LIN {X 0,Y 310.174,Z 752.952,A -85,B 0,C 180,E1 -16266.197,E2 -16266.197} C_VEL
LIN {X 0,Y 308.581,Z 766.008,A -85,B 0,C 180,E1 -16267.045,E2 -16267.045} C_VEL
LIN {X 0,Y 306.78,Z 778.403,A -85,B 0,C 180,E1 -16268.145,E2 -16268.145} C_VEL
LIN {X 0,Y 304.905,Z 789.628,A -85,B 0,C 180,E1 -16269.421,E2 -16269.421} C_VEL
LIN {X 0,Y 302.875,Z 800.82,A -85,B 0,C 180,E1 -16271.043,E2 -16271.043} C_VEL
LIN {X 0,Y 301.234,Z 810.089,A -85,B 0,C 180,E1 -16272.722,E2 -16272.722} C_VEL
LIN {X 0,Y 299.736,Z 818.952,A -85,B 0,C 180,E1 -16274.706,E2 -16274.706} C_VEL
LIN {X 0,Y 298.426,Z 826.179,A -85,B 0,C 180,E1 -16276.726,E2 -16276.726} C_VEL
LIN {X 0,Y 297.408,Z 832.88,A -85,B 0,C 180,E1 -16279.103,E2 -16279.103} C_VEL
LIN {X 0,Y 297.02,Z 837.35,A -85,B 0,C 180,E1 -16281.153,E2 -16281.153} C_VEL
LIN {X 0,Y 296.852,Z 840.748,A -85,B 0,C 180,E1 -16283.202,E2 -16283.202} C_VEL
LIN {X 0,Y 296.856,Z 842.474,A -85,B 0,C 180,E1 -16284.566,E2 -16284.566} C_VEL
LIN {X 0,Y 296.874,Z 843.732,A -85,B 0,C 180,E1 -16285.928,E2 -16285.928} C_VEL
LIN {X 0,Y 297.025,Z 844.574,A -85,B 0,C 180,E1 -16287.288,E2 -16287.288} C_VEL
LIN {X 0,Y 297.158,Z 845.011,A -85,B 0,C 180,E1 -16288.645,E2 -16288.645} C_VEL
LIN {X 0,Y 297.234,Z 845.034,A -85,B 0,C 180,E1 -16290,E2 -16290} C_VEL
LIN {X 0,Y 297.191,Z 844.583,A -85,B 0,C 180,E1 -16291.355,E2 -16291.355} C_VEL
LIN {X 0,Y 296.924,Z 842.624,A -85,B 0,C 180,E1 -16294.072,E2 -16294.072} C_VEL
LIN {X 0,Y 296.873,Z 840.823,A -85,B 0,C 180,E1 -16296.128,E2 -16296.128} C_VEL
LIN {X 0,Y 296.997,Z 836.98,A -85,B 0,C 180,E1 -16298.848,E2 -16298.848} C_VEL
LIN {X 0,Y 297.414,Z 832.866,A -85,B 0,C 180,E1 -16300.897,E2 -16300.897} C_VEL
LIN {X 0,Y 298.462,Z 826.576,A -85,B 0,C 180,E1 -16303.272,E2 -16303.272} C_VEL
LIN {X 0,Y 299.734,Z 819.761,A -85,B 0,C 180,E1 -16305.294,E2 -16305.294} C_VEL
LIN {X 0,Y 301.187,Z 811.484,A -85,B 0,C 180,E1 -16307.273,E2 -16307.273} C_VEL
LIN {X 0,Y 302.982,Z 802.663,A -85,B 0,C 180,E1 -16308.95,E2 -16308.95} C_VEL
LIN {X 0,Y 305.047,Z 792.026,A -85,B 0,C 180,E1 -16310.569,E2 -16310.569} C_VEL
LIN {X 0,Y 306.884,Z 781.465,A -85,B 0,C 180,E1 -16311.847,E2 -16311.847} C_VEL
LIN {X 0,Y 308.764,Z 769.655,A -85,B 0,C 180,E1 -16312.941,E2 -16312.941} C_VEL
LIN {X 0,Y 310.313,Z 757.416,A -85,B 0,C 180,E1 -16313.791,E2 -16313.791} C_VEL
LIN {X 0,Y 311.486,Z 744.997,A -85,B 0,C 180,E1 -16314.397,E2 -16314.397} C_VEL
LIN {X 0,Y 312.109,Z 730.684,A -85,B 0,C 180,E1 -16314.824,E2 -16314.824} C_VEL
LIN {X 0,Y 313.469,Z 680.173,A -85,B 0,C 180,E1 -16316,E2 -16316} C_VEL
LIN {X 0,Y 310.399,Z 651.031,A -85,B 0,C 180,E1 -16317.095,E2 -16317.095} C_VEL
LIN {X 0,Y 306.302,Z 623.478,A -85,B 0,C 180,E1 -16318.301,E2 -16318.301} C_VEL
LIN {X 0,Y 305.071,Z 620.075,A -85,B 0,C 180,E1 -16318.539,E2 -16318.539} C_VEL
LIN {X 0,Y 303.666,Z 615.782,A -85,B 0,C 180,E1 -16318.956,E2 -16318.956} C_VEL
LIN {X 0,Y 300.127,Z 600.639,A -85,B 0,C 180,E1 -16322.586,E2 -16322.586} C_VEL
LIN {X 0,Y 298.408,Z 593.316,A -85,B 0,C 180,E1 -16324.418,E2 -16324.418} C_VEL
LIN {X 0,Y 298.438,Z 593.306,A -85,B 0,C 180,E1 -16327.753,E2 -16327.753} C_VEL
LIN {X 0,Y 298.418,Z 593.307,A -85,B 0,C 180,E1 -16331.255,E2 -16331.255} C_VEL
LIN {X 0,Y 298.414,Z 593.308,A -85,B 0,C 180,E1 -16334.952,E2 -16334.952} C_VEL
LIN {X 0,Y 298.448,Z 593.306,A -85,B 0,C 180,E1 -16338.749,E2 -16338.749} C_VEL
LIN {X 0,Y 298.466,Z 593.305,A -85,B 0,C 180,E1 -16343.185,E2 -16343.185} C_VEL
LIN {X 0,Y 298.393,Z 593.313,A -85,B 0,C 180,E1 -16347.199,E2 -16347.199} C_VEL
LIN {X 0,Y 298.427,Z 593.294,A -85,B 0,C 180,E1 -16350.614,E2 -16350.614} C_VEL
LIN {X 0,Y 298.479,Z 593.303,A -85,B 0,C 180,E1 -16353.474,E2 -16353.474} C_VEL
LIN {X 0,Y 298.428,Z 593.291,A -85,B 0,C 180,E1 -16356.697,E2 -16356.697} C_VEL
LIN {X 0,Y 298.533,Z 593.299,A -85,B 0,C 180,E1 -16360.756,E2 -16360.756} C_VEL
LIN {X 0,Y 298.586,Z 593.274,A -85,B 0,C 180,E1 -16364.994,E2 -16364.994} C_VEL
LIN {X 0,Y 298.584,Z 593.283,A -85,B 0,C 180,E1 -16369.146,E2 -16369.146} C_VEL
LIN {X 0,Y 298.734,Z 593.253,A -85,B 0,C 180,E1 -16371.885,E2 -16371.885} C_VEL
LIN {X 0,Y 298.654,Z 593.285,A -85,B 0,C 180,E1 -16374.599,E2 -16374.599} C_VEL
LIN {X 0,Y 298.918,Z 593.227,A -85,B 0,C 180,E1 -16378.653,E2 -16378.653} C_VEL
LIN {X 0,Y 298.92,Z 593.25,A -85,B 0,C 180,E1 -16381.347,E2 -16381.347} C_VEL
LIN {X 0,Y 298.652,Z 593.259,A -85,B 0,C 180,E1 -16385.401,E2 -16385.401} C_VEL
LIN {X 0,Y 298.748,Z 593.267,A -85,B 0,C 180,E1 -16388.114,E2 -16388.114} C_VEL
LIN {X 0,Y 298.545,Z 593.277,A -85,B 0,C 180,E1 -16392.232,E2 -16392.232} C_VEL
LIN {X 0,Y 298.6,Z 593.291,A -85,B 0,C 180,E1 -16395.209,E2 -16395.209} C_VEL
LIN {X 0,Y 298.533,Z 593.282,A -85,B 0,C 180,E1 -16399.244,E2 -16399.244} C_VEL
LIN {X 0,Y 298.451,Z 593.299,A -85,B 0,C 180,E1 -16403.598,E2 -16403.598} C_VEL
LIN {X 0,Y 298.484,Z 593.301,A -85,B 0,C 180,E1 -16406.575,E2 -16406.575} C_VEL
LIN {X 0,Y 298.417,Z 593.299,A -85,B 0,C 180,E1 -16409.642,E2 -16409.642} C_VEL
LIN {X 0,Y 298.393,Z 593.316,A -85,B 0,C 180,E1 -16412.801,E2 -16412.801} C_VEL
LIN {X 0,Y 298.461,Z 593.309,A -85,B 0,C 180,E1 -16416.813,E2 -16416.813} C_VEL
LIN {X 0,Y 298.414,Z 593.286,A -85,B 0,C 180,E1 -16421.095,E2 -16421.095} C_VEL
LIN {X 0,Y 298.385,Z 593.317,A -85,B 0,C 180,E1 -16424.959,E2 -16424.959} C_VEL
LIN {X 0,Y 298.384,Z 593.301,A -85,B 0,C 180,E1 -16428.826,E2 -16428.826} C_VEL
LIN {X 0,Y 299.45,Z 596.241,A -85,B 0,C 180,E1 -16429.063,E2 -16429.063} C_VEL
LIN {X 0,Y 300.765,Z 598.211,A -85,B 0,C 180,E1 -16429.286,E2 -16429.286} C_VEL
LIN {X 0,Y 309.42,Z 613.922,A -85,B 0,C 180,E1 -16430.763,E2 -16430.763} C_VEL
LIN {X 0,Y 315.519,Z 626.227,A -85,B 0,C 180,E1 -16431.769,E2 -16431.769} C_VEL
LIN {X 0,Y 313.772,Z 685.154,A -85,B 0,C 180,E1 -16433.117,E2 -16433.117} C_VEL
LIN {X 0,Y 313.31,Z 698.588,A -85,B 0,C 180,E1 -16433.58,E2 -16433.58} C_VEL
LIN {X 0,Y 312.556,Z 710.365,A -85,B 0,C 180,E1 -16434.225,E2 -16434.225} C_VEL
LIN {X 0,Y 311.19,Z 723.672,A -85,B 0,C 180,E1 -16435.233,E2 -16435.233} C_VEL
LIN {X 0,Y 309.686,Z 735.273,A -85,B 0,C 180,E1 -16436.417,E2 -16436.417} C_VEL
LIN {X 0,Y 307.85,Z 746.627,A -85,B 0,C 180,E1 -16437.903,E2 -16437.903} C_VEL
LIN {X 0,Y 306.244,Z 755.192,A -85,B 0,C 180,E1 -16439.296,E2 -16439.296} C_VEL
LIN {X 0,Y 304.567,Z 763.776,A -85,B 0,C 180,E1 -16441.016,E2 -16441.016} C_VEL
LIN {X 0,Y 302.719,Z 772.004,A -85,B 0,C 180,E1 -16443.083,E2 -16443.083} C_VEL
LIN {X 0,Y 301.166,Z 778.564,A -85,B 0,C 180,E1 -16445.163,E2 -16445.163} C_VEL
LIN {X 0,Y 299.918,Z 783.703,A -85,B 0,C 180,E1 -16447.255,E2 -16447.255} C_VEL
LIN {X 0,Y 298.942,Z 787.596,A -85,B 0,C 180,E1 -16449.351,E2 -16449.351} C_VEL
LIN {X 0,Y 298.401,Z 789.563,A -85,B 0,C 180,E1 -16450.748,E2 -16450.748} C_VEL
LIN {X 0,Y 297.93,Z 791.107,A -85,B 0,C 180,E1 -16452.142,E2 -16452.142} C_VEL
LIN {X 0,Y 297.608,Z 792.207,A -85,B 0,C 180,E1 -16453.538,E2 -16453.538} C_VEL
LIN {X 0,Y 297.279,Z 793.073,A -85,B 0,C 180,E1 -16455.763,E2 -16455.763} C_VEL
LIN {X 0,Y 297.101,Z 792.993,A -85,B 0,C 180,E1 -16457.708,E2 -16457.708} C_VEL
LIN {X 0,Y 297.138,Z 791.447,A -85,B 0,C 180,E1 -16460.47,E2 -16460.47} C_VEL
LIN {X 0,Y 297.472,Z 788.763,A -85,B 0,C 180,E1 -16462.878,E2 -16462.878} C_VEL
LIN {X 0,Y 297.889,Z 784.726,A -85,B 0,C 180,E1 -16465.264,E2 -16465.264} C_VEL
LIN {X 0,Y 298.386,Z 780.095,A -85,B 0,C 180,E1 -16467.3,E2 -16467.3} C_VEL
LIN {X 0,Y 299.358,Z 773.121,A -85,B 0,C 180,E1 -16469.664,E2 -16469.664} C_VEL
LIN {X 0,Y 300.322,Z 765.523,A -85,B 0,C 180,E1 -16471.676,E2 -16471.676} C_VEL
LIN {X 0,Y 301.652,Z 756.013,A -85,B 0,C 180,E1 -16473.673,E2 -16473.673} C_VEL
LIN {X 0,Y 302.841,Z 746.175,A -85,B 0,C 180,E1 -16475.326,E2 -16475.326} C_VEL
LIN {X 0,Y 304.074,Z 735.11,A -85,B 0,C 180,E1 -16476.803,E2 -16476.803} C_VEL
LIN {X 0,Y 305.201,Z 724.278,A -85,B 0,C 180,E1 -16477.941,E2 -16477.941} C_VEL
LIN {X 0,Y 306.119,Z 712.245,A -85,B 0,C 180,E1 -16478.915,E2 -16478.915} C_VEL
LIN {X 0,Y 306.772,Z 699.048,A -85,B 0,C 180,E1 -16479.685,E2 -16479.685} C_VEL
LIN {X 0,Y 307.167,Z 685.86,A -85,B 0,C 180,E1 -16480.172,E2 -16480.172} C_VEL
LIN {X 0,Y 308.638,Z 618.658,A -85,B 0,C 180,E1 -16481.718,E2 -16481.718} C_VEL
LIN {X 0,Y 300.49,Z 598.313,A -85,B 0,C 180,E1 -16482.804,E2 -16482.804} C_VEL
LIN {X 0,Y 298.671,Z 593.897,A -85,B 0,C 180,E1 -16483.051,E2 -16483.051} C_VEL
LIN {X 0,Y 298.573,Z 593.291,A -85,B 0,C 180,E1 -16483.105,E2 -16483.105} C_VEL
LIN {X 0,Y 298.55,Z 593.296,A -85,B 0,C 180,E1 -16486.408,E2 -16486.408} C_VEL
LIN {X 0,Y 298.489,Z 593.302,A -85,B 0,C 180,E1 -16490.42,E2 -16490.42} C_VEL
LIN {X 0,Y 300.198,Z 597.98,A -85,B 0,C 180,E1 -16490.715,E2 -16490.715} C_VEL
LIN {X 0,Y 309.443,Z 620.601,A -85,B 0,C 180,E1 -16492.025,E2 -16492.025} C_VEL
LIN {X 0,Y 307.444,Z 689.886,A -85,B 0,C 180,E1 -16493.812,E2 -16493.812} C_VEL
LIN {X 0,Y 306.954,Z 703.275,A -85,B 0,C 180,E1 -16494.428,E2 -16494.428} C_VEL
LIN {X 0,Y 306.073,Z 716.586,A -85,B 0,C 180,E1 -16495.319,E2 -16495.319} C_VEL
LIN {X 0,Y 304.967,Z 729.092,A -85,B 0,C 180,E1 -16496.464,E2 -16496.464} C_VEL
LIN {X 0,Y 303.873,Z 739.878,A -85,B 0,C 180,E1 -16497.727,E2 -16497.727} C_VEL
LIN {X 0,Y 302.694,Z 749.874,A -85,B 0,C 180,E1 -16499.181,E2 -16499.181} C_VEL
LIN {X 0,Y 301.405,Z 759.749,A -85,B 0,C 180,E1 -16500.97,E2 -16500.97} C_VEL
LIN {X 0,Y 300.209,Z 763.729,A -85,B 0,C 180,E1 -16501.773,E2 -16501.773} C_VEL
LIN {X 0,Y 296.521,Z 769.833,A -85,B 0,C 180,E1 -16503.098,E2 -16503.098} C_VEL
LIN {X 0,Y 292.936,Z 775.382,A -85,B 0,C 180,E1 -16504.541,E2 -16504.541} C_VEL
LIN {X 0,Y 291.921,Z 778.388,A -85,B 0,C 180,E1 -16505.513,E2 -16505.513} C_VEL
LIN {X 0,Y 291.307,Z 782.87,A -85,B 0,C 180,E1 -16507.236,E2 -16507.236} C_VEL
LIN {X 0,Y 290.716,Z 787.192,A -85,B 0,C 180,E1 -16509.322,E2 -16509.322} C_VEL
LIN {X 0,Y 290.298,Z 790.365,A -85,B 0,C 180,E1 -16511.366,E2 -16511.366} C_VEL
LIN {X 0,Y 290.027,Z 792.549,A -85,B 0,C 180,E1 -16513.367,E2 -16513.367} C_VEL
LIN {X 0,Y 289.944,Z 793.863,A -85,B 0,C 180,E1 -16515.337,E2 -16515.337} C_VEL
LIN {X 0,Y 290.001,Z 794.378,A -85,B 0,C 180,E1 -16517.268,E2 -16517.268} C_VEL
LIN {X 0,Y 290.247,Z 794.094,A -85,B 0,C 180,E1 -16519.173,E2 -16519.173} C_VEL
LIN {X 0,Y 290.641,Z 793.064,A -85,B 0,C 180,E1 -16521.045,E2 -16521.045} C_VEL
LIN {X 0,Y 291.526,Z 790.21,A -85,B 0,C 180,E1 -16523.798,E2 -16523.798} C_VEL
LIN {X 0,Y 292.255,Z 787.193,A -85,B 0,C 180,E1 -16525.704,E2 -16525.704} C_VEL
LIN {X 0,Y 293.568,Z 781.749,A -85,B 0,C 180,E1 -16528.219,E2 -16528.219} C_VEL
LIN {X 0,Y 295.07,Z 775.583,A -85,B 0,C 180,E1 -16530.376,E2 -16530.376} C_VEL
LIN {X 0,Y 296.803,Z 767.866,A -85,B 0,C 180,E1 -16532.5,E2 -16532.5} C_VEL
LIN {X 0,Y 298.563,Z 759.264,A -85,B 0,C 180,E1 -16534.371,E2 -16534.371} C_VEL
LIN {X 0,Y 300.443,Z 749.499,A -85,B 0,C 180,E1 -16536.072,E2 -16536.072} C_VEL
LIN {X 0,Y 302.011,Z 739.942,A -85,B 0,C 180,E1 -16537.421,E2 -16537.421} C_VEL
LIN {X 0,Y 303.469,Z 729.502,A -85,B 0,C 180,E1 -16538.608,E2 -16538.608} C_VEL
LIN {X 0,Y 304.841,Z 717.293,A -85,B 0,C 180,E1 -16539.68,E2 -16539.68} C_VEL
LIN {X 0,Y 305.897,Z 703.764,A -85,B 0,C 180,E1 -16540.56,E2 -16540.56} C_VEL
LIN {X 0,Y 306.53,Z 690.829,A -85,B 0,C 180,E1 -16541.111,E2 -16541.111} C_VEL
LIN {X 0,Y 309.007,Z 627.426,A -85,B 0,C 180,E1 -16542.841,E2 -16542.841} C_VEL
LIN {X 0,Y 302.168,Z 613.302,A -85,B 0,C 180,E1 -16544.183,E2 -16544.183} C_VEL
LIN {X 0,Y 295.467,Z 601.572,A -85,B 0,C 180,E1 -16545.544,E2 -16545.544} C_VEL
LIN {X 0,Y 293.449,Z 598.204,A -85,B 0,C 180,E1 -16545.968,E2 -16545.968} C_VEL
LIN {X 0,Y 291.914,Z 595.837,A -85,B 0,C 180,E1 -16546.291,E2 -16546.291} C_VEL
LIN {X 0,Y 291.511,Z 594.173,A -85,B 0,C 180,E1 -16546.449,E2 -16546.449} C_VEL
LIN {X 0,Y 291.699,Z 594.15,A -85,B 0,C 180,E1 -16551.041,E2 -16551.041} C_VEL
LIN {X 0,Y 291.741,Z 594.143,A -85,B 0,C 180,E1 -16553.082,E2 -16553.082} C_VEL
LIN {X 0,Y 291.884,Z 594.126,A -85,B 0,C 180,E1 -16558.62,E2 -16558.62} C_VEL
LIN {X 0,Y 291.884,Z 594.126,A -85,B 0,C 180,E1 -16561.38,E2 -16561.38} C_VEL
LIN {X 0,Y 291.737,Z 594.136,A -85,B 0,C 180,E1 -16566.918,E2 -16566.918} C_VEL
LIN {X 0,Y 291.623,Z 594.149,A -85,B 0,C 180,E1 -16569.712,E2 -16569.712} C_VEL
LIN {X 0,Y 291.516,Z 594.158,A -85,B 0,C 180,E1 -16573.951,E2 -16573.951} C_VEL
LIN {X 0,Y 291.48,Z 594.163,A -85,B 0,C 180,E1 -16576.818,E2 -16576.818} C_VEL
LIN {X 0,Y 291.445,Z 594.172,A -85,B 0,C 180,E1 -16579.875,E2 -16579.875} C_VEL
LIN {X 0,Y 291.394,Z 594.179,A -85,B 0,C 180,E1 -16584.206,E2 -16584.206} C_VEL
LIN {X 0,Y 291.417,Z 594.176,A -85,B 0,C 180,E1 -16587.272,E2 -16587.272} C_VEL
LIN {X 0,Y 291.333,Z 594.19,A -85,B 0,C 180,E1 -16590.437,E2 -16590.437} C_VEL
LIN {X 0,Y 291.34,Z 594.188,A -85,B 0,C 180,E1 -16593.699,E2 -16593.699} C_VEL
LIN {X 0,Y 291.401,Z 594.185,A -85,B 0,C 180,E1 -16597.262,E2 -16597.262} C_VEL
LIN {X 0,Y 291.397,Z 594.188,A -85,B 0,C 180,E1 -16600.632,E2 -16600.632} C_VEL
LIN {X 0,Y 291.35,Z 594.193,A -85,B 0,C 180,E1 -16604.391,E2 -16604.391} C_VEL
LIN {X 0,Y 291.355,Z 594.195,A -85,B 0,C 180,E1 -16608.398,E2 -16608.398} C_VEL
LIN {X 0,Y 291.421,Z 594.36,A -85,B 0,C 180,E1 -16609.452,E2 -16609.452} C_VEL
LIN {X 0,Y 294.286,Z 604.468,A -85,B 0,C 180,E1 -16613.343,E2 -16613.343} C_VEL
LIN {X 0,Y 296.493,Z 613.544,A -85,B 0,C 180,E1 -16616.466,E2 -16616.466} C_VEL
LIN {X 0,Y 298.475,Z 623.474,A -85,B 0,C 180,E1 -16619.587,E2 -16619.587} C_VEL
LIN {X 0,Y 298.861,Z 626.642,A -85,B 0,C 180,E1 -16620.5,E2 -16620.5} C_VEL
LIN {X 0,Y 302.721,Z 646.5,A -85,B 0,C 180,E1 -16621.678,E2 -16621.678} C_VEL
LIN {X 0,Y 305.472,Z 665.59,A -85,B 0,C 180,E1 -16622.639,E2 -16622.639} C_VEL
LIN {X 0,Y 307.206,Z 685.196,A -85,B 0,C 180,E1 -16623.471,E2 -16623.471} C_VEL
LIN {X 0,Y 305.129,Z 738.474,A -85,B 0,C 180,E1 -16624.925,E2 -16624.925} C_VEL
LIN {X 0,Y 303.993,Z 752.145,A -85,B 0,C 180,E1 -16625.546,E2 -16625.546} C_VEL
LIN {X 0,Y 302.391,Z 764.748,A -85,B 0,C 180,E1 -16626.365,E2 -16626.365} C_VEL
LIN {X 0,Y 300.505,Z 777.257,A -85,B 0,C 180,E1 -16627.483,E2 -16627.483} C_VEL
LIN {X 0,Y 298.517,Z 788.54,A -85,B 0,C 180,E1 -16628.779,E2 -16628.779} C_VEL
LIN {X 0,Y 296.585,Z 798.8,A -85,B 0,C 180,E1 -16630.265,E2 -16630.265} C_VEL
LIN {X 0,Y 294.742,Z 808.126,A -85,B 0,C 180,E1 -16631.942,E2 -16631.942} C_VEL
LIN {X 0,Y 293.161,Z 817.32,A -85,B 0,C 180,E1 -16633.997,E2 -16633.997} C_VEL
LIN {X 0,Y 291.686,Z 824.774,A -85,B 0,C 180,E1 -16636.058,E2 -16636.058} C_VEL
LIN {X 0,Y 290.629,Z 830.768,A -85,B 0,C 180,E1 -16638.139,E2 -16638.139} C_VEL
LIN {X 0,Y 290.064,Z 835.554,A -85,B 0,C 180,E1 -16640.235,E2 -16640.235} C_VEL
LIN {X 0,Y 289.808,Z 839.251,A -85,B 0,C 180,E1 -16642.335,E2 -16642.335} C_VEL
LIN {X 0,Y 289.768,Z 841.932,A -85,B 0,C 180,E1 -16644.433,E2 -16644.433} C_VEL
LIN {X 0,Y 289.801,Z 843.156,A -85,B 0,C 180,E1 -16645.828,E2 -16645.828} C_VEL
LIN {X 0,Y 289.931,Z 843.978,A -85,B 0,C 180,E1 -16647.221,E2 -16647.221} C_VEL
LIN {X 0,Y 290.095,Z 844.397,A -85,B 0,C 180,E1 -16648.612,E2 -16648.612} C_VEL
LIN {X 0,Y 290.169,Z 844.386,A -85,B 0,C 180,E1 -16650,E2 -16650} C_VEL
LIN {X 0,Y 290.13,Z 843.902,A -85,B 0,C 180,E1 -16651.388,E2 -16651.388} C_VEL
LIN {X 0,Y 289.847,Z 842.072,A -85,B 0,C 180,E1 -16654.171,E2 -16654.171} C_VEL
LIN {X 0,Y 289.782,Z 840.523,A -85,B 0,C 180,E1 -16656.085,E2 -16656.085} C_VEL
LIN {X 0,Y 289.846,Z 837.625,A -85,B 0,C 180,E1 -16658.365,E2 -16658.365} C_VEL
LIN {X 0,Y 290.201,Z 833.917,A -85,B 0,C 180,E1 -16660.465,E2 -16660.465} C_VEL
LIN {X 0,Y 290.962,Z 829.105,A -85,B 0,C 180,E1 -16662.555,E2 -16662.555} C_VEL
LIN {X 0,Y 292.076,Z 823.047,A -85,B 0,C 180,E1 -16664.634,E2 -16664.634} C_VEL
LIN {X 0,Y 293.602,Z 815.546,A -85,B 0,C 180,E1 -16666.693,E2 -16666.693} C_VEL
LIN {X 0,Y 295.098,Z 807.922,A -85,B 0,C 180,E1 -16668.394,E2 -16668.394} C_VEL
LIN {X 0,Y 297.092,Z 798.69,A -85,B 0,C 180,E1 -16670.06,E2 -16670.06} C_VEL
LIN {X 0,Y 299.166,Z 788.43,A -85,B 0,C 180,E1 -16671.534,E2 -16671.534} C_VEL
LIN {X 0,Y 301.092,Z 777.083,A -85,B 0,C 180,E1 -16672.833,E2 -16672.833} C_VEL
LIN {X 0,Y 302.962,Z 765.224,A -85,B 0,C 180,E1 -16673.86,E2 -16673.86} C_VEL
LIN {X 0,Y 304.544,Z 752.108,A -85,B 0,C 180,E1 -16674.679,E2 -16674.679} C_VEL
LIN {X 0,Y 305.53,Z 739.137,A -85,B 0,C 180,E1 -16675.23,E2 -16675.23} C_VEL
LIN {X 0,Y 307.314,Z 681.287,A -85,B 0,C 180,E1 -16676.624,E2 -16676.624} C_VEL
LIN {X 0,Y 304.371,Z 652.431,A -85,B 0,C 180,E1 -16677.736,E2 -16677.736} C_VEL
LIN {X 0,Y 300.371,Z 625.297,A -85,B 0,C 180,E1 -16678.96,E2 -16678.96} C_VEL
LIN {X 0,Y 297.016,Z 617.029,A -85,B 0,C 180,E1 -16679.655,E2 -16679.655} C_VEL
LIN {X 0,Y 295.814,Z 613.256,A -85,B 0,C 180,E1 -16680.069,E2 -16680.069} C_VEL
LIN {X 0,Y 292.608,Z 599.303,A -85,B 0,C 180,E1 -16683.533,E2 -16683.533} C_VEL
LIN {X 0,Y 291.357,Z 594.192,A -85,B 0,C 180,E1 -16684.902,E2 -16684.902} C_VEL
LIN {X 0,Y 291.398,Z 594.187,A -85,B 0,C 180,E1 -16687.259,E2 -16687.259} C_VEL
LIN {X 0,Y 291.375,Z 594.188,A -85,B 0,C 180,E1 -16690.634,E2 -16690.634} C_VEL
LIN {X 0,Y 291.35,Z 594.191,A -85,B 0,C 180,E1 -16694.389,E2 -16694.389} C_VEL
LIN {X 0,Y 291.383,Z 594.188,A -85,B 0,C 180,E1 -16698.39,E2 -16698.39} C_VEL
LIN {X 0,Y 291.381,Z 594.18,A -85,B 0,C 180,E1 -16701.163,E2 -16701.163} C_VEL
LIN {X 0,Y 291.382,Z 594.175,A -85,B 0,C 180,E1 -16704.629,E2 -16704.629} C_VEL
LIN {X 0,Y 291.371,Z 594.19,A -85,B 0,C 180,E1 -16707.95,E2 -16707.95} C_VEL
LIN {X 0,Y 291.377,Z 594.17,A -85,B 0,C 180,E1 -16711.158,E2 -16711.158} C_VEL
LIN {X 0,Y 291.412,Z 594.188,A -85,B 0,C 180,E1 -16714.271,E2 -16714.271} C_VEL
LIN {X 0,Y 291.375,Z 594.167,A -85,B 0,C 180,E1 -16717.299,E2 -16717.299} C_VEL
LIN {X 0,Y 291.452,Z 594.18,A -85,B 0,C 180,E1 -16720.27,E2 -16720.27} C_VEL
LIN {X 0,Y 291.534,Z 594.149,A -85,B 0,C 180,E1 -16724.634,E2 -16724.634} C_VEL
LIN {X 0,Y 291.528,Z 594.164,A -85,B 0,C 180,E1 -16728.88,E2 -16728.88} C_VEL
LIN {X 0,Y 291.681,Z 594.129,A -85,B 0,C 180,E1 -16731.688,E2 -16731.688} C_VEL
LIN {X 0,Y 291.624,Z 594.159,A -85,B 0,C 180,E1 -16734.468,E2 -16734.468} C_VEL
LIN {X 0,Y 291.884,Z 594.103,A -85,B 0,C 180,E1 -16738.62,E2 -16738.62} C_VEL
LIN {X 0,Y 291.886,Z 594.126,A -85,B 0,C 180,E1 -16741.38,E2 -16741.38} C_VEL
LIN {X 0,Y 291.735,Z 594.128,A -85,B 0,C 180,E1 -16746.918,E2 -16746.918} C_VEL
LIN {X 0,Y 291.622,Z 594.157,A -85,B 0,C 180,E1 -16749.712,E2 -16749.712} C_VEL
LIN {X 0,Y 291.514,Z 594.163,A -85,B 0,C 180,E1 -16753.951,E2 -16753.951} C_VEL
LIN {X 0,Y 291.48,Z 594.173,A -85,B 0,C 180,E1 -16756.818,E2 -16756.818} C_VEL
LIN {X 0,Y 291.445,Z 594.169,A -85,B 0,C 180,E1 -16759.875,E2 -16759.875} C_VEL
LIN {X 0,Y 291.394,Z 594.173,A -85,B 0,C 180,E1 -16764.206,E2 -16764.206} C_VEL
LIN {X 0,Y 291.417,Z 594.187,A -85,B 0,C 180,E1 -16767.272,E2 -16767.272} C_VEL
LIN {X 0,Y 291.334,Z 594.183,A -85,B 0,C 180,E1 -16770.437,E2 -16770.437} C_VEL
LIN {X 0,Y 291.341,Z 594.185,A -85,B 0,C 180,E1 -16773.699,E2 -16773.699} C_VEL
LIN {X 0,Y 291.394,Z 594.186,A -85,B 0,C 180,E1 -16777.26,E2 -16777.26} C_VEL
LIN {X 0,Y 291.373,Z 594.169,A -85,B 0,C 180,E1 -16780.636,E2 -16780.636} C_VEL
LIN {X 0,Y 291.32,Z 594.19,A -85,B 0,C 180,E1 -16784.396,E2 -16784.396} C_VEL
LIN {X 0,Y 291.33,Z 594.186,A -85,B 0,C 180,E1 -16787.928,E2 -16787.928} C_VEL
LIN {X 0,Y 292.414,Z 597.171,A -85,B 0,C 180,E1 -16788.165,E2 -16788.165} C_VEL
LIN {X 0,Y 293.785,Z 599.206,A -85,B 0,C 180,E1 -16788.41,E2 -16788.41} C_VEL
LIN {X 0,Y 301.771,Z 613.273,A -85,B 0,C 180,E1 -16789.834,E2 -16789.834} C_VEL
LIN {X 0,Y 309.06,Z 627.626,A -85,B 0,C 180,E1 -16791.09,E2 -16791.09} C_VEL
LIN {X 0,Y 309.369,Z 628.292,A -85,B 0,C 180,E1 -16791.143,E2 -16791.143} C_VEL
LIN {X 0,Y 307.578,Z 686.482,A -85,B 0,C 180,E1 -16792.501,E2 -16792.501} C_VEL
LIN {X 0,Y 307.049,Z 699.861,A -85,B 0,C 180,E1 -16792.983,E2 -16792.983} C_VEL
LIN {X 0,Y 306.191,Z 712.162,A -85,B 0,C 180,E1 -16793.688,E2 -16793.688} C_VEL
LIN {X 0,Y 304.919,Z 724.057,A -85,B 0,C 180,E1 -16794.616,E2 -16794.616} C_VEL
LIN {X 0,Y 303.353,Z 735.709,A -85,B 0,C 180,E1 -16795.819,E2 -16795.819} C_VEL
LIN {X 0,Y 301.436,Z 747.126,A -85,B 0,C 180,E1 -16797.339,E2 -16797.339} C_VEL
LIN {X 0,Y 299.554,Z 756.65,A -85,B 0,C 180,E1 -16798.926,E2 -16798.926} C_VEL
LIN {X 0,Y 297.601,Z 765.965,A -85,B 0,C 180,E1 -16800.901,E2 -16800.901} C_VEL
LIN {X 0,Y 295.881,Z 773.155,A -85,B 0,C 180,E1 -16802.792,E2 -16802.792} C_VEL
LIN {X 0,Y 294.505,Z 778.613,A -85,B 0,C 180,E1 -16804.562,E2 -16804.562} C_VEL
LIN {X 0,Y 293.17,Z 783.876,A -85,B 0,C 180,E1 -16806.701,E2 -16806.701} C_VEL
LIN {X 0,Y 292.088,Z 787.892,A -85,B 0,C 180,E1 -16808.844,E2 -16808.844} C_VEL
LIN {X 0,Y 291.507,Z 789.927,A -85,B 0,C 180,E1 -16810.274,E2 -16810.274} C_VEL
LIN {X 0,Y 291,Z 791.516,A -85,B 0,C 180,E1 -16811.702,E2 -16811.702} C_VEL
LIN {X 0,Y 290.619,Z 792.691,A -85,B 0,C 180,E1 -16813.131,E2 -16813.131} C_VEL
LIN {X 0,Y 290.248,Z 793.677,A -85,B 0,C 180,E1 -16815.593,E2 -16815.593} C_VEL
LIN {X 0,Y 290.043,Z 793.633,A -85,B 0,C 180,E1 -16817.404,E2 -16817.404} C_VEL
LIN {X 0,Y 289.983,Z 793.14,A -85,B 0,C 180,E1 -16818.821,E2 -16818.821} C_VEL
LIN {X 0,Y 290.062,Z 792.211,A -85,B 0,C 180,E1 -16820.235,E2 -16820.235} C_VEL
LIN {X 0,Y 290.386,Z 789.39,A -85,B 0,C 180,E1 -16822.883,E2 -16822.883} C_VEL
LIN {X 0,Y 290.79,Z 785.722,A -85,B 0,C 180,E1 -16825.148,E2 -16825.148} C_VEL
LIN {X 0,Y 291.297,Z 781.194,A -85,B 0,C 180,E1 -16827.234,E2 -16827.234} C_VEL
LIN {X 0,Y 292.258,Z 774.336,A -85,B 0,C 180,E1 -16829.656,E2 -16829.656} C_VEL
LIN {X 0,Y 293.241,Z 766.927,A -85,B 0,C 180,E1 -16831.717,E2 -16831.717} C_VEL
LIN {X 0,Y 294.607,Z 757.576,A -85,B 0,C 180,E1 -16833.761,E2 -16833.761} C_VEL
LIN {X 0,Y 295.834,Z 747.984,A -85,B 0,C 180,E1 -16835.453,E2 -16835.453} C_VEL
LIN {X 0,Y 297.092,Z 737.087,A -85,B 0,C 180,E1 -16836.98,E2 -16836.98} C_VEL
LIN {X 0,Y 298.335,Z 725.579,A -85,B 0,C 180,E1 -16838.243,E2 -16838.243} C_VEL
LIN {X 0,Y 299.275,Z 714.259,A -85,B 0,C 180,E1 -16839.206,E2 -16839.206} C_VEL
LIN {X 0,Y 299.971,Z 701.612,A -85,B 0,C 180,E1 -16839.992,E2 -16839.992} C_VEL
LIN {X 0,Y 300.403,Z 688.428,A -85,B 0,C 180,E1 -16840.531,E2 -16840.531} C_VEL
LIN {X 0,Y 301.938,Z 620.18,A -85,B 0,C 180,E1 -16842.148,E2 -16842.148} C_VEL
LIN {X 0,Y 292.562,Z 597.064,A -85,B 0,C 180,E1 -16843.438,E2 -16843.438} C_VEL
LIN {X 0,Y 291.527,Z 594.176,A -85,B 0,C 180,E1 -16843.595,E2 -16843.595} C_VEL
LIN {X 0,Y 291.489,Z 594.176,A -85,B 0,C 180,E1 -16846.817,E2 -16846.817} C_VEL
LIN {X 0,Y 291.477,Z 594.34,A -85,B 0,C 180,E1 -16849.932,E2 -16849.932} C_VEL
LIN {X 0,Y 294.223,Z 601.329,A -85,B 0,C 180,E1 -16850.355,E2 -16850.355} C_VEL
LIN {X 0,Y 302.776,Z 622.373,A -85,B 0,C 180,E1 -16851.599,E2 -16851.599} C_VEL
LIN {X 0,Y 300.774,Z 689.567,A -85,B 0,C 180,E1 -16853.367,E2 -16853.367} C_VEL
LIN {X 0,Y 300.206,Z 703.239,A -85,B 0,C 180,E1 -16853.992,E2 -16853.992} C_VEL
LIN {X 0,Y 299.353,Z 716.315,A -85,B 0,C 180,E1 -16854.87,E2 -16854.87} C_VEL
LIN {X 0,Y 298.284,Z 728.201,A -85,B 0,C 180,E1 -16855.953,E2 -16855.953} C_VEL
LIN {X 0,Y 297.155,Z 739.462,A -85,B 0,C 180,E1 -16857.273,E2 -16857.273} C_VEL
LIN {X 0,Y 295.831,Z 750.148,A -85,B 0,C 180,E1 -16858.833,E2 -16858.833} C_VEL
LIN {X 0,Y 294.668,Z 758.79,A -85,B 0,C 180,E1 -16860.395,E2 -16860.395} C_VEL
LIN {X 0,Y 293.411,Z 767.581,A -85,B 0,C 180,E1 -16862.348,E2 -16862.348} C_VEL
LIN {X 0,Y 292.398,Z 774.694,A -85,B 0,C 180,E1 -16864.303,E2 -16864.303} C_VEL
LIN {X 0,Y 291.921,Z 778.388,A -85,B 0,C 180,E1 -16865.513,E2 -16865.513} C_VEL
LIN {X 0,Y 290.946,Z 781.212,A -85,B 0,C 180,E1 -16866.515,E2 -16866.515} C_VEL
LIN {X 0,Y 287.56,Z 785.41,A -85,B 0,C 180,E1 -16868.167,E2 -16868.167} C_VEL
LIN {X 0,Y 284.739,Z 788.247,A -85,B 0,C 180,E1 -16869.551,E2 -16869.551} C_VEL
LIN {X 0,Y 283.432,Z 790.041,A -85,B 0,C 180,E1 -16870.663,E2 -16870.663} C_VEL
LIN {X 0,Y 283.269,Z 790.561,A -85,B 0,C 180,E1 -16871.049,E2 -16871.049} C_VEL
LIN {X 0,Y 282.906,Z 793.603,A -85,B 0,C 180,E1 -16873.91,E2 -16873.91} C_VEL
LIN {X 0,Y 282.87,Z 794.772,A -85,B 0,C 180,E1 -16876.095,E2 -16876.095} C_VEL
LIN {X 0,Y 283.05,Z 794.987,A -85,B 0,C 180,E1 -16878.148,E2 -16878.148} C_VEL
LIN {X 0,Y 283.396,Z 794.351,A -85,B 0,C 180,E1 -16880.242,E2 -16880.242} C_VEL
LIN {X 0,Y 283.969,Z 792.801,A -85,B 0,C 180,E1 -16882.368,E2 -16882.368} C_VEL
LIN {X 0,Y 284.722,Z 790.243,A -85,B 0,C 180,E1 -16884.542,E2 -16884.542} C_VEL
LIN {X 0,Y 285.725,Z 786.547,A -85,B 0,C 180,E1 -16886.749,E2 -16886.749} C_VEL
LIN {X 0,Y 287.074,Z 781.354,A -85,B 0,C 180,E1 -16889.062,E2 -16889.062} C_VEL
LIN {X 0,Y 288.663,Z 775.063,A -85,B 0,C 180,E1 -16891.218,E2 -16891.218} C_VEL
LIN {X 0,Y 290.268,Z 768.174,A -85,B 0,C 180,E1 -16893.099,E2 -16893.099} C_VEL
LIN {X 0,Y 292.236,Z 759.109,A -85,B 0,C 180,E1 -16895.08,E2 -16895.08} C_VEL
LIN {X 0,Y 294.2,Z 749.333,A -85,B 0,C 180,E1 -16896.786,E2 -16896.786} C_VEL
LIN {X 0,Y 296.058,Z 738.242,A -85,B 0,C 180,E1 -16898.326,E2 -16898.326} C_VEL
LIN {X 0,Y 297.656,Z 726.811,A -85,B 0,C 180,E1 -16899.577,E2 -16899.577} C_VEL
LIN {X 0,Y 299.051,Z 714.666,A -85,B 0,C 180,E1 -16900.585,E2 -16900.585} C_VEL
LIN {X 0,Y 299.994,Z 701.118,A -85,B 0,C 180,E1 -16901.408,E2 -16901.408} C_VEL
LIN {X 0,Y 300.568,Z 689.478,A -85,B 0,C 180,E1 -16901.864,E2 -16901.864} C_VEL
LIN {X 0,Y 303.02,Z 629.485,A -85,B 0,C 180,E1 -16903.528,E2 -16903.528} C_VEL
LIN {X 0,Y 296.467,Z 616.134,A -85,B 0,C 180,E1 -16904.885,E2 -16904.885} C_VEL
LIN {X 0,Y 288.962,Z 603.117,A -85,B 0,C 180,E1 -16906.489,E2 -16906.489} C_VEL
LIN {X 0,Y 286.585,Z 599.306,A -85,B 0,C 180,E1 -16907.024,E2 -16907.024} C_VEL
LIN {X 0,Y 284.926,Z 596.775,A -85,B 0,C 180,E1 -16907.4,E2 -16907.4} C_VEL
LIN {X 0,Y 284.472,Z 595.052,A -85,B 0,C 180,E1 -16907.606,E2 -16907.606} C_VEL
LIN {X 0,Y 284.653,Z 595.029,A -85,B 0,C 180,E1 -16911.481,E2 -16911.481} C_VEL
LIN {X 0,Y 284.597,Z 595.033,A -85,B 0,C 180,E1 -16914.331,E2 -16914.331} C_VEL
LIN {X 0,Y 284.85,Z 595.002,A -85,B 0,C 180,E1 -16918.586,E2 -16918.586} C_VEL
LIN {X 0,Y 284.85,Z 595.002,A -85,B 0,C 180,E1 -16921.414,E2 -16921.414} C_VEL
LIN {X 0,Y 284.689,Z 595.014,A -85,B 0,C 180,E1 -16927.09,E2 -16927.09} C_VEL
LIN {X 0,Y 284.561,Z 595.028,A -85,B 0,C 180,E1 -16929.956,E2 -16929.956} C_VEL
LIN {X 0,Y 284.472,Z 595.037,A -85,B 0,C 180,E1 -16934.303,E2 -16934.303} C_VEL
LIN {X 0,Y 284.419,Z 595.043,A -85,B 0,C 180,E1 -16937.249,E2 -16937.249} C_VEL
LIN {X 0,Y 284.373,Z 595.051,A -85,B 0,C 180,E1 -16940.243,E2 -16940.243} C_VEL
LIN {X 0,Y 284.363,Z 595.054,A -85,B 0,C 180,E1 -16943.876,E2 -16943.876} C_VEL
LIN {X 0,Y 284.392,Z 595.052,A -85,B 0,C 180,E1 -16947.174,E2 -16947.174} C_VEL
LIN {X 0,Y 284.291,Z 595.068,A -85,B 0,C 180,E1 -16951.275,E2 -16951.275} C_VEL
LIN {X 0,Y 284.358,Z 595.065,A -85,B 0,C 180,E1 -16955.355,E2 -16955.355} C_VEL
LIN {X 0,Y 284.332,Z 595.069,A -85,B 0,C 180,E1 -16958.166,E2 -16958.166} C_VEL
LIN {X 0,Y 284.337,Z 595.064,A -85,B 0,C 180,E1 -16962.141,E2 -16962.141} C_VEL
LIN {X 0,Y 284.315,Z 595.07,A -85,B 0,C 180,E1 -16966.202,E2 -16966.202} C_VEL
LIN {X 0,Y 284.308,Z 595.077,A -85,B 0,C 180,E1 -16968.317,E2 -16968.317} C_VEL
LIN {X 0,Y 286.345,Z 601.99,A -85,B 0,C 180,E1 -16971.196,E2 -16971.196} C_VEL
LIN {X 0,Y 288.806,Z 611.27,A -85,B 0,C 180,E1 -16974.674,E2 -16974.674} C_VEL
LIN {X 0,Y 290.87,Z 620.758,A -85,B 0,C 180,E1 -16977.89,E2 -16977.89} C_VEL
LIN {X 0,Y 291.865,Z 625.981,A -85,B 0,C 180,E1 -16979.475,E2 -16979.475} C_VEL
LIN {X 0,Y 293.782,Z 631.344,A -85,B 0,C 180,E1 -16979.948,E2 -16979.948} C_VEL
LIN {X 0,Y 297.711,Z 653.297,A -85,B 0,C 180,E1 -16981.256,E2 -16981.256} C_VEL
LIN {X 0,Y 299.726,Z 668.87,A -85,B 0,C 180,E1 -16982.034,E2 -16982.034} C_VEL
LIN {X 0,Y 301.208,Z 685.376,A -85,B 0,C 180,E1 -16982.761,E2 -16982.761} C_VEL
LIN {X 0,Y 299.004,Z 737.652,A -85,B 0,C 180,E1 -16984.226,E2 -16984.226} C_VEL
LIN {X 0,Y 297.826,Z 751.399,A -85,B 0,C 180,E1 -16984.865,E2 -16984.865} C_VEL
LIN {X 0,Y 296.26,Z 763.463,A -85,B 0,C 180,E1 -16985.659,E2 -16985.659} C_VEL
LIN {X 0,Y 294.269,Z 776.113,A -85,B 0,C 180,E1 -16986.793,E2 -16986.793} C_VEL
LIN {X 0,Y 292.174,Z 787.482,A -85,B 0,C 180,E1 -16988.11,E2 -16988.11} C_VEL
LIN {X 0,Y 290.109,Z 797.832,A -85,B 0,C 180,E1 -16989.621,E2 -16989.621} C_VEL
LIN {X 0,Y 287.988,Z 808.049,A -85,B 0,C 180,E1 -16991.504,E2 -16991.504} C_VEL
LIN {X 0,Y 286.264,Z 817.387,A -85,B 0,C 180,E1 -16993.669,E2 -16993.669} C_VEL
LIN {X 0,Y 284.73,Z 824.451,A -85,B 0,C 180,E1 -16995.71,E2 -16995.71} C_VEL
LIN {X 0,Y 283.657,Z 830.372,A -85,B 0,C 180,E1 -16997.843,E2 -16997.843} C_VEL
LIN {X 0,Y 283.03,Z 835.104,A -85,B 0,C 180,E1 -16999.99,E2 -16999.99} C_VEL
LIN {X 0,Y 282.735,Z 838.751,A -85,B 0,C 180,E1 -17002.142,E2 -17002.142} C_VEL
LIN {X 0,Y 282.699,Z 841.39,A -85,B 0,C 180,E1 -17004.293,E2 -17004.293} C_VEL
LIN {X 0,Y 282.729,Z 842.587,A -85,B 0,C 180,E1 -17005.723,E2 -17005.723} C_VEL
LIN {X 0,Y 282.838,Z 843.383,A -85,B 0,C 180,E1 -17007.152,E2 -17007.152} C_VEL
LIN {X 0,Y 283.032,Z 843.783,A -85,B 0,C 180,E1 -17008.577,E2 -17008.577} C_VEL
LIN {X 0,Y 283.106,Z 843.726,A -85,B 0,C 180,E1 -17010,E2 -17010} C_VEL
LIN {X 0,Y 283.068,Z 843.218,A -85,B 0,C 180,E1 -17011.423,E2 -17011.423} C_VEL
LIN {X 0,Y 282.699,Z 840.483,A -85,B 0,C 180,E1 -17015.707,E2 -17015.707} C_VEL
LIN {X 0,Y 282.676,Z 839.047,A -85,B 0,C 180,E1 -17017.141,E2 -17017.141} C_VEL
LIN {X 0,Y 282.878,Z 836.06,A -85,B 0,C 180,E1 -17019.293,E2 -17019.293} C_VEL
LIN {X 0,Y 283.362,Z 832.046,A -85,B 0,C 180,E1 -17021.444,E2 -17021.444} C_VEL
LIN {X 0,Y 284.603,Z 825.919,A -85,B 0,C 180,E1 -17023.931,E2 -17023.931} C_VEL
LIN {X 0,Y 285.977,Z 819.391,A -85,B 0,C 180,E1 -17026.003,E2 -17026.003} C_VEL
LIN {X 0,Y 287.637,Z 810.972,A -85,B 0,C 180,E1 -17028.151,E2 -17028.151} C_VEL
LIN {X 0,Y 289.559,Z 802.546,A -85,B 0,C 180,E1 -17029.864,E2 -17029.864} C_VEL
LIN {X 0,Y 291.807,Z 792.151,A -85,B 0,C 180,E1 -17031.548,E2 -17031.548} C_VEL
LIN {X 0,Y 294.073,Z 780.481,A -85,B 0,C 180,E1 -17033.038,E2 -17033.038} C_VEL
LIN {X 0,Y 296.065,Z 768.773,A -85,B 0,C 180,E1 -17034.172,E2 -17034.172} C_VEL
LIN {X 0,Y 297.739,Z 756.652,A -85,B 0,C 180,E1 -17035.049,E2 -17035.049} C_VEL
LIN {X 0,Y 299.021,Z 744.322,A -85,B 0,C 180,E1 -17035.679,E2 -17035.679} C_VEL
LIN {X 0,Y 299.71,Z 730.208,A -85,B 0,C 180,E1 -17036.129,E2 -17036.129} C_VEL
LIN {X 0,Y 301.158,Z 681.548,A -85,B 0,C 180,E1 -17037.304,E2 -17037.304} C_VEL
LIN {X 0,Y 298.433,Z 654.367,A -85,B 0,C 180,E1 -17038.381,E2 -17038.381} C_VEL
LIN {X 0,Y 294.638,Z 627.928,A -85,B 0,C 180,E1 -17039.606,E2 -17039.606} C_VEL
LIN {X 0,Y 289.849,Z 616.104,A -85,B 0,C 180,E1 -17040.634,E2 -17040.634} C_VEL
LIN {X 0,Y 287.924,Z 610.439,A -85,B 0,C 180,E1 -17041.315,E2 -17041.315} C_VEL
LIN {X 0,Y 284.61,Z 596.367,A -85,B 0,C 180,E1 -17044.956,E2 -17044.956} C_VEL
LIN {X 0,Y 284.337,Z 595.067,A -85,B 0,C 180,E1 -17045.346,E2 -17045.346} C_VEL
LIN {X 0,Y 284.328,Z 595.061,A -85,B 0,C 180,E1 -17048.165,E2 -17048.165} C_VEL
LIN {X 0,Y 284.302,Z 595.062,A -85,B 0,C 180,E1 -17051.869,E2 -17051.869} C_VEL
LIN {X 0,Y 284.305,Z 595.06,A -85,B 0,C 180,E1 -17055.796,E2 -17055.796} C_VEL
LIN {X 0,Y 284.336,Z 595.069,A -85,B 0,C 180,E1 -17058.136,E2 -17058.136} C_VEL
LIN {X 0,Y 284.342,Z 595.065,A -85,B 0,C 180,E1 -17062.271,E2 -17062.271} C_VEL
LIN {X 0,Y 284.319,Z 595.051,A -85,B 0,C 180,E1 -17065.352,E2 -17065.352} C_VEL
LIN {X 0,Y 284.294,Z 595.07,A -85,B 0,C 180,E1 -17068.725,E2 -17068.725} C_VEL
LIN {X 0,Y 284.392,Z 595.054,A -85,B 0,C 180,E1 -17072.826,E2 -17072.826} C_VEL
LIN {X 0,Y 284.36,Z 595.043,A -85,B 0,C 180,E1 -17076.706,E2 -17076.706} C_VEL
LIN {X 0,Y 284.397,Z 595.057,A -85,B 0,C 180,E1 -17081.261,E2 -17081.261} C_VEL
LIN {X 0,Y 284.472,Z 595.028,A -85,B 0,C 180,E1 -17084.469,E2 -17084.469} C_VEL
LIN {X 0,Y 284.48,Z 595.044,A -85,B 0,C 180,E1 -17088.601,E2 -17088.601} C_VEL
LIN {X 0,Y 284.632,Z 595.005,A -85,B 0,C 180,E1 -17091.48,E2 -17091.48} C_VEL
LIN {X 0,Y 284.594,Z 595.034,A -85,B 0,C 180,E1 -17094.331,E2 -17094.331} C_VEL
LIN {X 0,Y 284.85,Z 594.978,A -85,B 0,C 180,E1 -17098.586,E2 -17098.586} C_VEL
LIN {X 0,Y 284.852,Z 595.002,A -85,B 0,C 180,E1 -17101.414,E2 -17101.414} C_VEL
LIN {X 0,Y 284.687,Z 595.008,A -85,B 0,C 180,E1 -17107.09,E2 -17107.09} C_VEL
LIN {X 0,Y 284.56,Z 595.037,A -85,B 0,C 180,E1 -17109.956,E2 -17109.956} C_VEL
LIN {X 0,Y 284.475,Z 595.042,A -85,B 0,C 180,E1 -17114.303,E2 -17114.303} C_VEL
LIN {X 0,Y 284.419,Z 595.048,A -85,B 0,C 180,E1 -17117.249,E2 -17117.249} C_VEL
LIN {X 0,Y 284.373,Z 595.053,A -85,B 0,C 180,E1 -17120.243,E2 -17120.243} C_VEL
LIN {X 0,Y 284.363,Z 595.051,A -85,B 0,C 180,E1 -17123.875,E2 -17123.875} C_VEL
LIN {X 0,Y 284.392,Z 595.062,A -85,B 0,C 180,E1 -17127.174,E2 -17127.174} C_VEL
LIN {X 0,Y 284.293,Z 595.067,A -85,B 0,C 180,E1 -17131.275,E2 -17131.275} C_VEL
LIN {X 0,Y 284.357,Z 595.057,A -85,B 0,C 180,E1 -17135.355,E2 -17135.355} C_VEL
LIN {X 0,Y 284.325,Z 595.067,A -85,B 0,C 180,E1 -17138.167,E2 -17138.167} C_VEL
LIN {X 0,Y 284.298,Z 595.037,A -85,B 0,C 180,E1 -17141.871,E2 -17141.871} C_VEL
LIN {X 0,Y 284.266,Z 595.065,A -85,B 0,C 180,E1 -17146.193,E2 -17146.193} C_VEL
LIN {X 0,Y 284.298,Z 595.233,A -85,B 0,C 180,E1 -17146.963,E2 -17146.963} C_VEL
LIN {X 0,Y 285.312,Z 597.937,A -85,B 0,C 180,E1 -17147.193,E2 -17147.193} C_VEL
LIN {X 0,Y 286.807,Z 600.146,A -85,B 0,C 180,E1 -17147.475,E2 -17147.475} C_VEL
LIN {X 0,Y 295.875,Z 615.839,A -85,B 0,C 180,E1 -17149.166,E2 -17149.166} C_VEL
LIN {X 0,Y 303.283,Z 630.387,A -85,B 0,C 180,E1 -17150.491,E2 -17150.491} C_VEL
LIN {X 0,Y 301.407,Z 688.29,A -85,B 0,C 180,E1 -17151.869,E2 -17151.869} C_VEL
LIN {X 0,Y 300.821,Z 701.559,A -85,B 0,C 180,E1 -17152.383,E2 -17152.383} C_VEL
LIN {X 0,Y 299.873,Z 714.233,A -85,B 0,C 180,E1 -17153.149,E2 -17153.149} C_VEL
LIN {X 0,Y 298.463,Z 726.337,A -85,B 0,C 180,E1 -17154.146,E2 -17154.146} C_VEL
LIN {X 0,Y 296.821,Z 737.579,A -85,B 0,C 180,E1 -17155.372,E2 -17155.372} C_VEL
LIN {X 0,Y 294.999,Z 747.809,A -85,B 0,C 180,E1 -17156.775,E2 -17156.775} C_VEL
LIN {X 0,Y 293.287,Z 756.177,A -85,B 0,C 180,E1 -17158.186,E2 -17158.186} C_VEL
LIN {X 0,Y 291.287,Z 765.422,A -85,B 0,C 180,E1 -17160.12,E2 -17160.12} C_VEL
LIN {X 0,Y 289.366,Z 773.078,A -85,B 0,C 180,E1 -17162.126,E2 -17162.126} C_VEL
LIN {X 0,Y 287.461,Z 780.253,A -85,B 0,C 180,E1 -17164.513,E2 -17164.513} C_VEL
LIN {X 0,Y 286.023,Z 785.545,A -85,B 0,C 180,E1 -17166.85,E2 -17166.85} C_VEL
LIN {X 0,Y 284.896,Z 789.379,A -85,B 0,C 180,E1 -17169.117,E2 -17169.117} C_VEL
LIN {X 0,Y 284.095,Z 791.928,A -85,B 0,C 180,E1 -17171.241,E2 -17171.241} C_VEL
LIN {X 0,Y 283.659,Z 793.149,A -85,B 0,C 180,E1 -17172.704,E2 -17172.704} C_VEL
LIN {X 0,Y 283.201,Z 794.284,A -85,B 0,C 180,E1 -17175.429,E2 -17175.429} C_VEL
LIN {X 0,Y 283.005,Z 794.265,A -85,B 0,C 180,E1 -17177.086,E2 -17177.086} C_VEL
LIN {X 0,Y 282.907,Z 793.843,A -85,B 0,C 180,E1 -17178.537,E2 -17178.537} C_VEL
LIN {X 0,Y 282.967,Z 792.975,A -85,B 0,C 180,E1 -17179.988,E2 -17179.988} C_VEL
LIN {X 0,Y 283.309,Z 790.027,A -85,B 0,C 180,E1 -17182.875,E2 -17182.875} C_VEL
LIN {X 0,Y 283.676,Z 786.679,A -85,B 0,C 180,E1 -17185.026,E2 -17185.026} C_VEL
LIN {X 0,Y 284.205,Z 782.265,A -85,B 0,C 180,E1 -17187.165,E2 -17187.165} C_VEL
LIN {X 0,Y 285.159,Z 775.539,A -85,B 0,C 180,E1 -17189.647,E2 -17189.647} C_VEL
LIN {X 0,Y 286.156,Z 768.263,A -85,B 0,C 180,E1 -17191.759,E2 -17191.759} C_VEL
LIN {X 0,Y 287.296,Z 760.811,A -85,B 0,C 180,E1 -17193.506,E2 -17193.506} C_VEL
LIN {X 0,Y 288.686,Z 750.745,A -85,B 0,C 180,E1 -17195.413,E2 -17195.413} C_VEL
LIN {X 0,Y 289.924,Z 740.553,A -85,B 0,C 180,E1 -17196.961,E2 -17196.961} C_VEL
LIN {X 0,Y 291.257,Z 729.175,A -85,B 0,C 180,E1 -17198.324,E2 -17198.324} C_VEL
LIN {X 0,Y 292.364,Z 717.175,A -85,B 0,C 180,E1 -17199.425,E2 -17199.425} C_VEL
LIN {X 0,Y 293.154,Z 704.147,A -85,B 0,C 180,E1 -17200.314,E2 -17200.314} C_VEL
LIN {X 0,Y 293.666,Z 690.766,A -85,B 0,C 180,E1 -17200.907,E2 -17200.907} C_VEL
LIN {X 0,Y 295.255,Z 621.677,A -85,B 0,C 180,E1 -17202.596,E2 -17202.596} C_VEL
LIN {X 0,Y 286.417,Z 600.118,A -85,B 0,C 180,E1 -17203.849,E2 -17203.849} C_VEL
LIN {X 0,Y 284.515,Z 595.199,A -85,B 0,C 180,E1 -17204.137,E2 -17204.137} C_VEL
LIN {X 0,Y 284.428,Z 595.056,A -85,B 0,C 180,E1 -17207.248,E2 -17207.248} C_VEL
LIN {X 0,Y 284.438,Z 595.151,A -85,B 0,C 180,E1 -17209.391,E2 -17209.391} C_VEL
LIN {X 0,Y 286.334,Z 600.141,A -85,B 0,C 180,E1 -17209.697,E2 -17209.697} C_VEL
LIN {X 0,Y 296.098,Z 623.759,A -85,B 0,C 180,E1 -17211.157,E2 -17211.157} C_VEL
LIN {X 0,Y 293.983,Z 690.893,A -85,B 0,C 180,E1 -17212.975,E2 -17212.975} C_VEL
LIN {X 0,Y 293.456,Z 704.04,A -85,B 0,C 180,E1 -17213.602,E2 -17213.602} C_VEL
LIN {X 0,Y 292.525,Z 717.316,A -85,B 0,C 180,E1 -17214.519,E2 -17214.519} C_VEL
LIN {X 0,Y 291.349,Z 730.075,A -85,B 0,C 180,E1 -17215.734,E2 -17215.734} C_VEL
LIN {X 0,Y 290.081,Z 741.812,A -85,B 0,C 180,E1 -17217.176,E2 -17217.176} C_VEL
LIN {X 0,Y 288.711,Z 752.226,A -85,B 0,C 180,E1 -17218.796,E2 -17218.796} C_VEL
LIN {X 0,Y 287.365,Z 762.058,A -85,B 0,C 180,E1 -17220.698,E2 -17220.698} C_VEL
LIN {X 0,Y 286.113,Z 770.408,A -85,B 0,C 180,E1 -17222.71,E2 -17222.71} C_VEL
LIN {X 0,Y 285.032,Z 777.947,A -85,B 0,C 180,E1 -17225.006,E2 -17225.006} C_VEL
LIN {X 0,Y 284.317,Z 783.18,A -85,B 0,C 180,E1 -17227.01,E2 -17227.01} C_VEL
LIN {X 0,Y 283.73,Z 787.327,A -85,B 0,C 180,E1 -17229.011,E2 -17229.011} C_VEL
LIN {X 0,Y 283.269,Z 790.561,A -85,B 0,C 180,E1 -17231.049,E2 -17231.049} C_VEL
LIN {X 0,Y 282.409,Z 792.052,A -85,B 0,C 180,E1 -17232.197,E2 -17232.197} C_VEL
LIN {X 0,Y 279.352,Z 794.011,A -85,B 0,C 180,E1 -17234.08,E2 -17234.08} C_VEL
LIN {X 0,Y 276.905,Z 795.073,A -85,B 0,C 180,E1 -17235.625,E2 -17235.625} C_VEL
LIN {X 0,Y 275.927,Z 795.531,A -85,B 0,C 180,E1 -17236.834,E2 -17236.834} C_VEL
LIN {X 0,Y 275.881,Z 795.591,A -85,B 0,C 180,E1 -17237.243,E2 -17237.243} C_VEL
LIN {X 0,Y 276.224,Z 795.331,A -85,B 0,C 180,E1 -17239.754,E2 -17239.754} C_VEL
LIN {X 0,Y 276.937,Z 793.622,A -85,B 0,C 180,E1 -17242.478,E2 -17242.478} C_VEL
LIN {X 0,Y 277.608,Z 791.587,A -85,B 0,C 180,E1 -17244.389,E2 -17244.389} C_VEL
LIN {X 0,Y 278.953,Z 787.005,A -85,B 0,C 180,E1 -17247.252,E2 -17247.252} C_VEL
LIN {X 0,Y 280.173,Z 782.52,A -85,B 0,C 180,E1 -17249.305,E2 -17249.305} C_VEL
LIN {X 0,Y 282.017,Z 775.651,A -85,B 0,C 180,E1 -17251.739,E2 -17251.739} C_VEL
LIN {X 0,Y 283.983,Z 767.611,A -85,B 0,C 180,E1 -17253.942,E2 -17253.942} C_VEL
LIN {X 0,Y 286.09,Z 758.591,A -85,B 0,C 180,E1 -17255.905,E2 -17255.905} C_VEL
LIN {X 0,Y 288.191,Z 748.418,A -85,B 0,C 180,E1 -17257.655,E2 -17257.655} C_VEL
LIN {X 0,Y 289.972,Z 738.033,A -85,B 0,C 180,E1 -17259.091,E2 -17259.091} C_VEL
LIN {X 0,Y 291.688,Z 726.37,A -85,B 0,C 180,E1 -17260.36,E2 -17260.36} C_VEL
LIN {X 0,Y 293.11,Z 713.816,A -85,B 0,C 180,E1 -17261.385,E2 -17261.385} C_VEL
LIN {X 0,Y 294.034,Z 700.621,A -85,B 0,C 180,E1 -17262.178,E2 -17262.178} C_VEL
LIN {X 0,Y 294.636,Z 688.332,A -85,B 0,C 180,E1 -17262.637,E2 -17262.637} C_VEL
LIN {X 0,Y 297.179,Z 631.967,A -85,B 0,C 180,E1 -17264.227,E2 -17264.227} C_VEL
LIN {X 0,Y 291.468,Z 620.251,A -85,B 0,C 180,E1 -17265.468,E2 -17265.468} C_VEL
LIN {X 0,Y 284.575,Z 608.041,A -85,B 0,C 180,E1 -17267.023,E2 -17267.023} C_VEL
LIN {X 0,Y 281.623,Z 603.544,A -85,B 0,C 180,E1 -17267.701,E2 -17267.701} C_VEL
LIN {X 0,Y 279.656,Z 600.269,A -85,B 0,C 180,E1 -17268.178,E2 -17268.178} C_VEL
LIN {X 0,Y 277.91,Z 597.73,A -85,B 0,C 180,E1 -17268.605,E2 -17268.605} C_VEL
LIN {X 0,Y 277.463,Z 595.922,A -85,B 0,C 180,E1 -17268.772,E2 -17268.772} C_VEL
LIN {X 0,Y 277.61,Z 595.906,A -85,B 0,C 180,E1 -17271.263,E2 -17271.263} C_VEL
LIN {X 0,Y 277.568,Z 595.91,A -85,B 0,C 180,E1 -17274.187,E2 -17274.187} C_VEL
LIN {X 0,Y 277.816,Z 595.878,A -85,B 0,C 180,E1 -17278.55,E2 -17278.55} C_VEL
LIN {X 0,Y 277.816,Z 595.878,A -85,B 0,C 180,E1 -17281.45,E2 -17281.45} C_VEL
LIN {X 0,Y 277.644,Z 595.891,A -85,B 0,C 180,E1 -17287.271,E2 -17287.271} C_VEL
LIN {X 0,Y 277.501,Z 595.906,A -85,B 0,C 180,E1 -17290.212,E2 -17290.212} C_VEL
LIN {X 0,Y 277.422,Z 595.918,A -85,B 0,C 180,E1 -17294.675,E2 -17294.675} C_VEL
LIN {X 0,Y 277.34,Z 595.932,A -85,B 0,C 180,E1 -17299.234,E2 -17299.234} C_VEL
LIN {X 0,Y 277.313,Z 595.932,A -85,B 0,C 180,E1 -17304.171,E2 -17304.171} C_VEL
LIN {X 0,Y 277.321,Z 595.932,A -85,B 0,C 180,E1 -17307.506,E2 -17307.506} C_VEL
LIN {X 0,Y 277.268,Z 595.941,A -85,B 0,C 180,E1 -17310.482,E2 -17310.482} C_VEL
LIN {X 0,Y 277.25,Z 595.943,A -85,B 0,C 180,E1 -17313.895,E2 -17313.895} C_VEL
LIN {X 0,Y 277.286,Z 595.944,A -85,B 0,C 180,E1 -17317.466,E2 -17317.466} C_VEL
LIN {X 0,Y 277.261,Z 595.945,A -85,B 0,C 180,E1 -17321.227,E2 -17321.227} C_VEL
LIN {X 0,Y 277.247,Z 595.952,A -85,B 0,C 180,E1 -17325.217,E2 -17325.217} C_VEL
LIN {X 0,Y 277.277,Z 596.121,A -85,B 0,C 180,E1 -17327.213,E2 -17327.213} C_VEL
LIN {X 0,Y 279.682,Z 604.022,A -85,B 0,C 180,E1 -17330.698,E2 -17330.698} C_VEL
LIN {X 0,Y 282.026,Z 612.874,A -85,B 0,C 180,E1 -17334.155,E2 -17334.155} C_VEL
LIN {X 0,Y 283.969,Z 621.792,A -85,B 0,C 180,E1 -17337.296,E2 -17337.296} C_VEL
LIN {X 0,Y 284.611,Z 625.021,A -85,B 0,C 180,E1 -17338.309,E2 -17338.309} C_VEL
LIN {X 0,Y 288.197,Z 633.534,A -85,B 0,C 180,E1 -17339.197,E2 -17339.197} C_VEL
LIN {X 0,Y 291.677,Z 653.396,A -85,B 0,C 180,E1 -17340.423,E2 -17340.423} C_VEL
LIN {X 0,Y 293.849,Z 670.329,A -85,B 0,C 180,E1 -17341.321,E2 -17341.321} C_VEL
LIN {X 0,Y 295.214,Z 686.434,A -85,B 0,C 180,E1 -17342.05,E2 -17342.05} C_VEL
LIN {X 0,Y 292.951,Z 737.341,A -85,B 0,C 180,E1 -17343.509,E2 -17343.509} C_VEL
LIN {X 0,Y 291.641,Z 751.683,A -85,B 0,C 180,E1 -17344.198,E2 -17344.198} C_VEL
LIN {X 0,Y 289.836,Z 764.417,A -85,B 0,C 180,E1 -17345.083,E2 -17345.083} C_VEL
LIN {X 0,Y 287.794,Z 776.675,A -85,B 0,C 180,E1 -17346.239,E2 -17346.239} C_VEL
LIN {X 0,Y 285.626,Z 787.778,A -85,B 0,C 180,E1 -17347.581,E2 -17347.581} C_VEL
LIN {X 0,Y 283.238,Z 798.865,A -85,B 0,C 180,E1 -17349.294,E2 -17349.294} C_VEL
LIN {X 0,Y 281.228,Z 807.977,A -85,B 0,C 180,E1 -17351.042,E2 -17351.042} C_VEL
LIN {X 0,Y 279.668,Z 815.896,A -85,B 0,C 180,E1 -17352.916,E2 -17352.916} C_VEL
LIN {X 0,Y 277.992,Z 823.081,A -85,B 0,C 180,E1 -17354.982,E2 -17354.982} C_VEL
LIN {X 0,Y 277.016,Z 828.207,A -85,B 0,C 180,E1 -17356.801,E2 -17356.801} C_VEL
LIN {X 0,Y 276.145,Z 833.245,A -85,B 0,C 180,E1 -17358.996,E2 -17358.996} C_VEL
LIN {X 0,Y 275.733,Z 837.175,A -85,B 0,C 180,E1 -17361.203,E2 -17361.203} C_VEL
LIN {X 0,Y 275.608,Z 839.246,A -85,B 0,C 180,E1 -17362.675,E2 -17362.675} C_VEL
LIN {X 0,Y 275.619,Z 840.843,A -85,B 0,C 180,E1 -17364.146,E2 -17364.146} C_VEL
LIN {X 0,Y 275.659,Z 842.019,A -85,B 0,C 180,E1 -17365.614,E2 -17365.614} C_VEL
LIN {X 0,Y 275.745,Z 842.792,A -85,B 0,C 180,E1 -17367.078,E2 -17367.078} C_VEL
LIN {X 0,Y 275.968,Z 843.162,A -85,B 0,C 180,E1 -17368.541,E2 -17368.541} C_VEL
LIN {X 0,Y 276.045,Z 843.058,A -85,B 0,C 180,E1 -17370,E2 -17370} C_VEL
LIN {X 0,Y 276.008,Z 842.524,A -85,B 0,C 180,E1 -17371.459,E2 -17371.459} C_VEL
LIN {X 0,Y 275.695,Z 840.97,A -85,B 0,C 180,E1 -17374.386,E2 -17374.386} C_VEL
LIN {X 0,Y 275.605,Z 839.828,A -85,B 0,C 180,E1 -17376.005,E2 -17376.005} C_VEL
LIN {X 0,Y 275.707,Z 836.701,A -85,B 0,C 180,E1 -17378.797,E2 -17378.797} C_VEL
LIN {X 0,Y 276.149,Z 833.094,A -85,B 0,C 180,E1 -17381.004,E2 -17381.004} C_VEL
LIN {X 0,Y 277.038,Z 828.398,A -85,B 0,C 180,E1 -17383.198,E2 -17383.198} C_VEL
LIN {X 0,Y 278.586,Z 821.339,A -85,B 0,C 180,E1 -17385.735,E2 -17385.735} C_VEL
LIN {X 0,Y 280.201,Z 813.741,A -85,B 0,C 180,E1 -17387.893,E2 -17387.893} C_VEL
LIN {X 0,Y 282.045,Z 806.011,A -85,B 0,C 180,E1 -17389.657,E2 -17389.657} C_VEL
LIN {X 0,Y 284.465,Z 795.525,A -85,B 0,C 180,E1 -17391.561,E2 -17391.561} C_VEL
LIN {X 0,Y 286.751,Z 784.882,A -85,B 0,C 180,E1 -17393.087,E2 -17393.087} C_VEL
LIN {X 0,Y 288.686,Z 774.578,A -85,B 0,C 180,E1 -17394.256,E2 -17394.256} C_VEL
LIN {X 0,Y 290.744,Z 762.218,A -85,B 0,C 180,E1 -17395.311,E2 -17395.311} C_VEL
LIN {X 0,Y 292.292,Z 750.002,A -85,B 0,C 180,E1 -17396.075,E2 -17396.075} C_VEL
LIN {X 0,Y 293.249,Z 737.722,A -85,B 0,C 180,E1 -17396.606,E2 -17396.606} C_VEL
LIN {X 0,Y 295.112,Z 682.598,A -85,B 0,C 180,E1 -17397.983,E2 -17397.983} C_VEL
LIN {X 0,Y 292.375,Z 654.888,A -85,B 0,C 180,E1 -17399.117,E2 -17399.117} C_VEL
LIN {X 0,Y 288.903,Z 630.56,A -85,B 0,C 180,E1 -17400.282,E2 -17400.282} C_VEL
LIN {X 0,Y 282.85,Z 615.614,A -85,B 0,C 180,E1 -17401.631,E2 -17401.631} C_VEL
LIN {X 0,Y 280.04,Z 607.749,A -85,B 0,C 180,E1 -17402.601,E2 -17402.601} C_VEL
LIN {X 0,Y 277.305,Z 595.944,A -85,B 0,C 180,E1 -17405.805,E2 -17405.805} C_VEL
LIN {X 0,Y 277.264,Z 595.944,A -85,B 0,C 180,E1 -17409.322,E2 -17409.322} C_VEL
LIN {X 0,Y 277.25,Z 595.948,A -85,B 0,C 180,E1 -17413.189,E2 -17413.189} C_VEL
LIN {X 0,Y 277.268,Z 595.945,A -85,B 0,C 180,E1 -17417.312,E2 -17417.312} C_VEL
LIN {X 0,Y 277.264,Z 595.935,A -85,B 0,C 180,E1 -17420.677,E2 -17420.677} C_VEL
LIN {X 0,Y 277.301,Z 595.93,A -85,B 0,C 180,E1 -17424.344,E2 -17424.344} C_VEL
LIN {X 0,Y 277.242,Z 595.949,A -85,B 0,C 180,E1 -17427.836,E2 -17427.836} C_VEL
LIN {X 0,Y 277.267,Z 595.927,A -85,B 0,C 180,E1 -17431.21,E2 -17431.21} C_VEL
LIN {X 0,Y 277.309,Z 595.942,A -85,B 0,C 180,E1 -17434.479,E2 -17434.479} C_VEL
LIN {X 0,Y 277.279,Z 595.923,A -85,B 0,C 180,E1 -17437.654,E2 -17437.654} C_VEL
LIN {X 0,Y 277.339,Z 595.939,A -85,B 0,C 180,E1 -17440.766,E2 -17440.766} C_VEL
LIN {X 0,Y 277.422,Z 595.912,A -85,B 0,C 180,E1 -17445.325,E2 -17445.325} C_VEL
LIN {X 0,Y 277.455,Z 595.908,A -85,B 0,C 180,E1 -17449.787,E2 -17449.787} C_VEL
LIN {X 0,Y 277.635,Z 595.887,A -85,B 0,C 180,E1 -17452.729,E2 -17452.729} C_VEL
LIN {X 0,Y 277.816,Z 595.854,A -85,B 0,C 180,E1 -17458.55,E2 -17458.55} C_VEL
LIN {X 0,Y 277.818,Z 595.878,A -85,B 0,C 180,E1 -17461.45,E2 -17461.45} C_VEL
LIN {X 0,Y 277.643,Z 595.887,A -85,B 0,C 180,E1 -17467.271,E2 -17467.271} C_VEL
LIN {X 0,Y 277.5,Z 595.917,A -85,B 0,C 180,E1 -17470.212,E2 -17470.212} C_VEL
LIN {X 0,Y 277.428,Z 595.922,A -85,B 0,C 180,E1 -17474.675,E2 -17474.675} C_VEL
LIN {X 0,Y 277.339,Z 595.92,A -85,B 0,C 180,E1 -17479.234,E2 -17479.234} C_VEL
LIN {X 0,Y 277.313,Z 595.927,A -85,B 0,C 180,E1 -17484.17,E2 -17484.17} C_VEL
LIN {X 0,Y 277.321,Z 595.941,A -85,B 0,C 180,E1 -17487.506,E2 -17487.506} C_VEL
LIN {X 0,Y 277.268,Z 595.935,A -85,B 0,C 180,E1 -17490.482,E2 -17490.482} C_VEL
LIN {X 0,Y 277.25,Z 595.939,A -85,B 0,C 180,E1 -17493.895,E2 -17493.895} C_VEL
LIN {X 0,Y 277.281,Z 595.943,A -85,B 0,C 180,E1 -17497.467,E2 -17497.467} C_VEL
LIN {X 0,Y 277.236,Z 595.92,A -85,B 0,C 180,E1 -17501.232,E2 -17501.232} C_VEL
LIN {X 0,Y 277.217,Z 595.956,A -85,B 0,C 180,E1 -17505.223,E2 -17505.223} C_VEL
LIN {X 0,Y 277.22,Z 595.947,A -85,B 0,C 180,E1 -17505.907,E2 -17505.907} C_VEL
LIN {X 0,Y 278.31,Z 598.924,A -85,B 0,C 180,E1 -17506.18,E2 -17506.18} C_VEL
LIN {X 0,Y 279.824,Z 601.036,A -85,B 0,C 180,E1 -17506.478,E2 -17506.478} C_VEL
LIN {X 0,Y 289.245,Z 617.051,A -85,B 0,C 180,E1 -17508.322,E2 -17508.322} C_VEL
LIN {X 0,Y 297.142,Z 632.372,A -85,B 0,C 180,E1 -17509.798,E2 -17509.798} C_VEL
LIN {X 0,Y 295.249,Z 690.885,A -85,B 0,C 180,E1 -17511.239,E2 -17511.239} C_VEL
LIN {X 0,Y 294.553,Z 704.666,A -85,B 0,C 180,E1 -17511.833,E2 -17511.833} C_VEL
LIN {X 0,Y 293.574,Z 716.599,A -85,B 0,C 180,E1 -17512.612,E2 -17512.612} C_VEL
LIN {X 0,Y 292.023,Z 728.529,A -85,B 0,C 180,E1 -17513.656,E2 -17513.656} C_VEL
LIN {X 0,Y 290.322,Z 739.38,A -85,B 0,C 180,E1 -17514.893,E2 -17514.893} C_VEL
LIN {X 0,Y 288.429,Z 749.477,A -85,B 0,C 180,E1 -17516.336,E2 -17516.336} C_VEL
LIN {X 0,Y 286.227,Z 759.468,A -85,B 0,C 180,E1 -17518.137,E2 -17518.137} C_VEL
LIN {X 0,Y 284.457,Z 767.119,A -85,B 0,C 180,E1 -17519.853,E2 -17519.853} C_VEL
LIN {X 0,Y 282.556,Z 774.238,A -85,B 0,C 180,E1 -17521.798,E2 -17521.798} C_VEL
LIN {X 0,Y 280.765,Z 780.591,A -85,B 0,C 180,E1 -17523.969,E2 -17523.969} C_VEL
LIN {X 0,Y 279.292,Z 785.764,A -85,B 0,C 180,E1 -17526.259,E2 -17526.259} C_VEL
LIN {X 0,Y 278.1,Z 789.593,A -85,B 0,C 180,E1 -17528.505,E2 -17528.505} C_VEL
LIN {X 0,Y 277.202,Z 792.34,A -85,B 0,C 180,E1 -17530.756,E2 -17530.756} C_VEL
LIN {X 0,Y 276.713,Z 793.607,A -85,B 0,C 180,E1 -17532.256,E2 -17532.256} C_VEL
LIN {X 0,Y 276.356,Z 794.47,A -85,B 0,C 180,E1 -17533.756,E2 -17533.756} C_VEL
LIN {X 0,Y 276.157,Z 794.891,A -85,B 0,C 180,E1 -17535.257,E2 -17535.257} C_VEL
LIN {X 0,Y 275.98,Z 794.897,A -85,B 0,C 180,E1 -17536.751,E2 -17536.751} C_VEL
LIN {X 0,Y 275.838,Z 794.52,A -85,B 0,C 180,E1 -17538.239,E2 -17538.239} C_VEL
LIN {X 0,Y 275.892,Z 793.736,A -85,B 0,C 180,E1 -17539.729,E2 -17539.729} C_VEL
LIN {X 0,Y 275.979,Z 792.509,A -85,B 0,C 180,E1 -17541.211,E2 -17541.211} C_VEL
LIN {X 0,Y 276.227,Z 790.657,A -85,B 0,C 180,E1 -17542.873,E2 -17542.873} C_VEL
LIN {X 0,Y 276.572,Z 787.619,A -85,B 0,C 180,E1 -17544.898,E2 -17544.898} C_VEL
LIN {X 0,Y 277.111,Z 783.302,A -85,B 0,C 180,E1 -17547.093,E2 -17547.093} C_VEL
LIN {X 0,Y 277.892,Z 777.803,A -85,B 0,C 180,E1 -17549.275,E2 -17549.275} C_VEL
LIN {X 0,Y 278.911,Z 770.904,A -85,B 0,C 180,E1 -17551.444,E2 -17551.444} C_VEL
LIN {X 0,Y 280.231,Z 762.282,A -85,B 0,C 180,E1 -17553.595,E2 -17553.595} C_VEL
LIN {X 0,Y 281.552,Z 753.454,A -85,B 0,C 180,E1 -17555.371,E2 -17555.371} C_VEL
LIN {X 0,Y 282.8,Z 743.745,A -85,B 0,C 180,E1 -17556.958,E2 -17556.958} C_VEL
LIN {X 0,Y 284.213,Z 732.099,A -85,B 0,C 180,E1 -17558.46,E2 -17558.46} C_VEL
LIN {X 0,Y 285.403,Z 720.103,A -85,B 0,C 180,E1 -17559.657,E2 -17559.657} C_VEL
LIN {X 0,Y 286.278,Z 707.138,A -85,B 0,C 180,E1 -17560.61,E2 -17560.61} C_VEL
LIN {X 0,Y 286.875,Z 694.299,A -85,B 0,C 180,E1 -17561.257,E2 -17561.257} C_VEL
LIN {X 0,Y 287.41,Z 671.704,A -85,B 0,C 180,E1 -17561.879,E2 -17561.879} C_VEL
LIN {X 0,Y 288.587,Z 623.301,A -85,B 0,C 180,E1 -17563.061,E2 -17563.061} C_VEL
LIN {X 0,Y 279.491,Z 601.155,A -85,B 0,C 180,E1 -17564.398,E2 -17564.398} C_VEL
LIN {X 0,Y 277.513,Z 596.327,A -85,B 0,C 180,E1 -17564.702,E2 -17564.702} C_VEL
LIN {X 0,Y 277.433,Z 595.927,A -85,B 0,C 180,E1 -17564.739,E2 -17564.739} C_VEL
LIN {X 0,Y 277.378,Z 595.934,A -85,B 0,C 180,E1 -17568.799,E2 -17568.799} C_VEL
LIN {X 0,Y 279.072,Z 600.54,A -85,B 0,C 180,E1 -17569.11,E2 -17569.11} C_VEL
LIN {X 0,Y 289.252,Z 624.983,A -85,B 0,C 180,E1 -17570.679,E2 -17570.679} C_VEL
LIN {X 0,Y 288.828,Z 642.247,A -85,B 0,C 180,E1 -17571.158,E2 -17571.158} C_VEL
LIN {X 0,Y 287.249,Z 692.044,A -85,B 0,C 180,E1 -17572.562,E2 -17572.562} C_VEL
LIN {X 0,Y 286.696,Z 705.515,A -85,B 0,C 180,E1 -17573.235,E2 -17573.235} C_VEL
LIN {X 0,Y 285.784,Z 717.571,A -85,B 0,C 180,E1 -17574.09,E2 -17574.09} C_VEL
LIN {X 0,Y 284.671,Z 729.272,A -85,B 0,C 180,E1 -17575.205,E2 -17575.205} C_VEL
LIN {X 0,Y 283.312,Z 741.729,A -85,B 0,C 180,E1 -17576.742,E2 -17576.742} C_VEL
LIN {X 0,Y 281.846,Z 752.615,A -85,B 0,C 180,E1 -17578.456,E2 -17578.456} C_VEL
LIN {X 0,Y 280.395,Z 762.938,A -85,B 0,C 180,E1 -17580.501,E2 -17580.501} C_VEL
LIN {X 0,Y 279.252,Z 770.308,A -85,B 0,C 180,E1 -17582.305,E2 -17582.305} C_VEL
LIN {X 0,Y 278.069,Z 778.006,A -85,B 0,C 180,E1 -17584.657,E2 -17584.657} C_VEL
LIN {X 0,Y 277.348,Z 783.185,A -85,B 0,C 180,E1 -17586.638,E2 -17586.638} C_VEL
LIN {X 0,Y 276.734,Z 787.53,A -85,B 0,C 180,E1 -17588.721,E2 -17588.721} C_VEL
LIN {X 0,Y 276.118,Z 791.7,A -85,B 0,C 180,E1 -17591.434,E2 -17591.434} C_VEL
LIN {X 0,Y 275.874,Z 793.797,A -85,B 0,C 180,E1 -17593.458,E2 -17593.458} C_VEL
LIN {X 0,Y 275.832,Z 795.481,A -85,B 0,C 180,E1 -17596.533,E2 -17596.533} C_VEL
LIN {X 0,Y 275.881,Z 795.591,A -85,B 0,C 180,E1 -17597.243,E2 -17597.243} C_VEL
LIN {X 0,Y 275.377,Z 795.731,A -85,B 0,C 180,E1 -17598.469,E2 -17598.469} C_VEL
LIN {X 0,Y 272.918,Z 795.57,A -85,B 0,C 180,E1 -17600.48,E2 -17600.48} C_VEL
LIN {X 0,Y 270.932,Z 794.851,A -85,B 0,C 180,E1 -17602.101,E2 -17602.101} C_VEL
LIN {X 0,Y 270.271,Z 793.824,A -85,B 0,C 180,E1 -17603.331,E2 -17603.331} C_VEL
LIN {X 0,Y 270.322,Z 793.37,A -85,B 0,C 180,E1 -17603.739,E2 -17603.739} C_VEL
LIN {X 0,Y 271.246,Z 790.496,A -85,B 0,C 180,E1 -17606.006,E2 -17606.006} C_VEL
LIN {X 0,Y 272.484,Z 786.394,A -85,B 0,C 180,E1 -17608.334,E2 -17608.334} C_VEL
LIN {X 0,Y 274.236,Z 780.441,A -85,B 0,C 180,E1 -17610.861,E2 -17610.861} C_VEL
LIN {X 0,Y 276.047,Z 773.933,A -85,B 0,C 180,E1 -17613.006,E2 -17613.006} C_VEL
LIN {X 0,Y 278.034,Z 766.325,A -85,B 0,C 180,E1 -17615.007,E2 -17615.007} C_VEL
LIN {X 0,Y 280.112,Z 757.495,A -85,B 0,C 180,E1 -17616.868,E2 -17616.868} C_VEL
LIN {X 0,Y 282.343,Z 746.908,A -85,B 0,C 180,E1 -17618.651,E2 -17618.651} C_VEL
LIN {X 0,Y 284.148,Z 736.691,A -85,B 0,C 180,E1 -17620.027,E2 -17620.027} C_VEL
LIN {X 0,Y 285.86,Z 724.913,A -85,B 0,C 180,E1 -17621.272,E2 -17621.272} C_VEL
LIN {X 0,Y 287.31,Z 712.259,A -85,B 0,C 180,E1 -17622.283,E2 -17622.283} C_VEL
LIN {X 0,Y 288.234,Z 699.503,A -85,B 0,C 180,E1 -17623.01,E2 -17623.01} C_VEL
LIN {X 0,Y 288.895,Z 684.62,A -85,B 0,C 180,E1 -17623.536,E2 -17623.536} C_VEL
LIN {X 0,Y 291.266,Z 634.033,A -85,B 0,C 180,E1 -17624.998,E2 -17624.998} C_VEL
LIN {X 0,Y 285.252,Z 621.797,A -85,B 0,C 180,E1 -17626.38,E2 -17626.38} C_VEL
LIN {X 0,Y 279.147,Z 611.311,A -85,B 0,C 180,E1 -17627.824,E2 -17627.824} C_VEL
LIN {X 0,Y 275.175,Z 605.007,A -85,B 0,C 180,E1 -17628.817,E2 -17628.817} C_VEL
LIN {X 0,Y 272.679,Z 601.154,A -85,B 0,C 180,E1 -17629.465,E2 -17629.465} C_VEL
LIN {X 0,Y 270.932,Z 598.581,A -85,B 0,C 180,E1 -17629.925,E2 -17629.925} C_VEL
LIN {X 0,Y 270.492,Z 596.789,A -85,B 0,C 180,E1 -17630.107,E2 -17630.107} C_VEL
LIN {X 0,Y 270.606,Z 596.774,A -85,B 0,C 180,E1 -17632.539,E2 -17632.539} C_VEL
LIN {X 0,Y 270.782,Z 596.753,A -85,B 0,C 180,E1 -17638.513,E2 -17638.513} C_VEL
LIN {X 0,Y 270.782,Z 596.754,A -85,B 0,C 180,E1 -17641.487,E2 -17641.487} C_VEL
LIN {X 0,Y 270.603,Z 596.769,A -85,B 0,C 180,E1 -17647.461,E2 -17647.461} C_VEL
LIN {X 0,Y 270.436,Z 596.786,A -85,B 0,C 180,E1 -17650.481,E2 -17650.481} C_VEL
LIN {X 0,Y 270.391,Z 596.798,A -85,B 0,C 180,E1 -17655.065,E2 -17655.065} C_VEL
LIN {X 0,Y 270.296,Z 596.806,A -85,B 0,C 180,E1 -17659.756,E2 -17659.756} C_VEL
LIN {X 0,Y 270.269,Z 596.811,A -85,B 0,C 180,E1 -17664.586,E2 -17664.586} C_VEL
LIN {X 0,Y 270.267,Z 596.812,A -85,B 0,C 180,E1 -17667.909,E2 -17667.909} C_VEL
LIN {X 0,Y 270.18,Z 596.826,A -85,B 0,C 180,E1 -17671.349,E2 -17671.349} C_VEL
LIN {X 0,Y 270.212,Z 596.827,A -85,B 0,C 180,E1 -17674.904,E2 -17674.904} C_VEL
LIN {X 0,Y 270.219,Z 596.822,A -85,B 0,C 180,E1 -17678.718,E2 -17678.718} C_VEL
LIN {X 0,Y 270.219,Z 596.826,A -85,B 0,C 180,E1 -17682.549,E2 -17682.549} C_VEL
LIN {X 0,Y 270.204,Z 596.909,A -85,B 0,C 180,E1 -17685.879,E2 -17685.879} C_VEL
LIN {X 0,Y 272.879,Z 605.501,A -85,B 0,C 180,E1 -17689.92,E2 -17689.92} C_VEL
LIN {X 0,Y 275.296,Z 614.665,A -85,B 0,C 180,E1 -17693.663,E2 -17693.663} C_VEL
LIN {X 0,Y 277.318,Z 623.993,A -85,B 0,C 180,E1 -17697.029,E2 -17697.029} C_VEL
LIN {X 0,Y 282.613,Z 635.9,A -85,B 0,C 180,E1 -17698.398,E2 -17698.398} C_VEL
LIN {X 0,Y 284.869,Z 647.909,A -85,B 0,C 180,E1 -17699.218,E2 -17699.218} C_VEL
LIN {X 0,Y 287.779,Z 668.547,A -85,B 0,C 180,E1 -17700.402,E2 -17700.402} C_VEL
LIN {X 0,Y 289.332,Z 687.501,A -85,B 0,C 180,E1 -17701.3,E2 -17701.3} C_VEL
LIN {X 0,Y 287.04,Z 735.987,A -85,B 0,C 180,E1 -17702.722,E2 -17702.722} C_VEL
LIN {X 0,Y 285.769,Z 749.782,A -85,B 0,C 180,E1 -17703.381,E2 -17703.381} C_VEL
LIN {X 0,Y 283.965,Z 762.415,A -85,B 0,C 180,E1 -17704.237,E2 -17704.237} C_VEL
LIN {X 0,Y 281.957,Z 774.148,A -85,B 0,C 180,E1 -17705.323,E2 -17705.323} C_VEL
LIN {X 0,Y 279.57,Z 785.591,A -85,B 0,C 180,E1 -17706.676,E2 -17706.676} C_VEL
LIN {X 0,Y 277.309,Z 796.012,A -85,B 0,C 180,E1 -17708.245,E2 -17708.245} C_VEL
LIN {X 0,Y 274.887,Z 806.294,A -85,B 0,C 180,E1 -17710.199,E2 -17710.199} C_VEL
LIN {X 0,Y 272.957,Z 815.09,A -85,B 0,C 180,E1 -17712.301,E2 -17712.301} C_VEL
LIN {X 0,Y 271.413,Z 821.671,A -85,B 0,C 180,E1 -17714.224,E2 -17714.224} C_VEL
LIN {X 0,Y 270.065,Z 827.894,A -85,B 0,C 180,E1 -17716.455,E2 -17716.455} C_VEL
LIN {X 0,Y 269.115,Z 832.867,A -85,B 0,C 180,E1 -17718.705,E2 -17718.705} C_VEL
LIN {X 0,Y 268.682,Z 836.734,A -85,B 0,C 180,E1 -17720.971,E2 -17720.971} C_VEL
LIN {X 0,Y 268.531,Z 838.749,A -85,B 0,C 180,E1 -17722.481,E2 -17722.481} C_VEL
LIN {X 0,Y 268.54,Z 840.306,A -85,B 0,C 180,E1 -17723.991,E2 -17723.991} C_VEL
LIN {X 0,Y 268.591,Z 841.456,A -85,B 0,C 180,E1 -17725.498,E2 -17725.498} C_VEL
LIN {X 0,Y 268.655,Z 842.201,A -85,B 0,C 180,E1 -17727.001,E2 -17727.001} C_VEL
LIN {X 0,Y 268.904,Z 842.527,A -85,B 0,C 180,E1 -17728.502,E2 -17728.502} C_VEL
LIN {X 0,Y 268.986,Z 842.392,A -85,B 0,C 180,E1 -17730,E2 -17730} C_VEL
LIN {X 0,Y 268.948,Z 841.832,A -85,B 0,C 180,E1 -17731.497,E2 -17731.497} C_VEL
LIN {X 0,Y 268.622,Z 840.42,A -85,B 0,C 180,E1 -17734.502,E2 -17734.502} C_VEL
LIN {X 0,Y 268.54,Z 839.425,A -85,B 0,C 180,E1 -17736.009,E2 -17736.009} C_VEL
LIN {X 0,Y 268.661,Z 836.237,A -85,B 0,C 180,E1 -17739.03,E2 -17739.03} C_VEL
LIN {X 0,Y 269.12,Z 832.678,A -85,B 0,C 180,E1 -17741.295,E2 -17741.295} C_VEL
LIN {X 0,Y 270.09,Z 828.044,A -85,B 0,C 180,E1 -17743.543,E2 -17743.543} C_VEL
LIN {X 0,Y 271.749,Z 821.056,A -85,B 0,C 180,E1 -17746.142,E2 -17746.142} C_VEL
LIN {X 0,Y 273.409,Z 813.527,A -85,B 0,C 180,E1 -17748.354,E2 -17748.354} C_VEL
LIN {X 0,Y 275.354,Z 805.886,A -85,B 0,C 180,E1 -17750.155,E2 -17750.155} C_VEL
LIN {X 0,Y 277.615,Z 796.614,A -85,B 0,C 180,E1 -17751.925,E2 -17751.925} C_VEL
LIN {X 0,Y 280.016,Z 786.323,A -85,B 0,C 180,E1 -17753.48,E2 -17753.48} C_VEL
LIN {X 0,Y 282.244,Z 774.937,A -85,B 0,C 180,E1 -17754.846,E2 -17754.846} C_VEL
LIN {X 0,Y 284.381,Z 762.971,A -85,B 0,C 180,E1 -17755.919,E2 -17755.919} C_VEL
LIN {X 0,Y 286.052,Z 750.488,A -85,B 0,C 180,E1 -17756.738,E2 -17756.738} C_VEL
LIN {X 0,Y 287.138,Z 737.687,A -85,B 0,C 180,E1 -17757.317,E2 -17757.317} C_VEL
LIN {X 0,Y 289.081,Z 683.406,A -85,B 0,C 180,E1 -17758.704,E2 -17758.704} C_VEL
LIN {X 0,Y 286.55,Z 656.867,A -85,B 0,C 180,E1 -17759.816,E2 -17759.816} C_VEL
LIN {X 0,Y 283.237,Z 633.156,A -85,B 0,C 180,E1 -17760.986,E2 -17760.986} C_VEL
LIN {X 0,Y 276.005,Z 615.606,A -85,B 0,C 180,E1 -17762.628,E2 -17762.628} C_VEL
LIN {X 0,Y 272.106,Z 604.646,A -85,B 0,C 180,E1 -17764.068,E2 -17764.068} C_VEL
LIN {X 0,Y 270.243,Z 596.823,A -85,B 0,C 180,E1 -17766.274,E2 -17766.274} C_VEL
LIN {X 0,Y 270.235,Z 596.822,A -85,B 0,C 180,E1 -17770.554,E2 -17770.554} C_VEL
LIN {X 0,Y 270.194,Z 596.825,A -85,B 0,C 180,E1 -17774.61,E2 -17774.61} C_VEL
LIN {X 0,Y 270.246,Z 596.818,A -85,B 0,C 180,E1 -17778.951,E2 -17778.951} C_VEL
LIN {X 0,Y 270.239,Z 596.821,A -85,B 0,C 180,E1 -17783.262,E2 -17783.262} C_VEL
LIN {X 0,Y 270.201,Z 596.82,A -85,B 0,C 180,E1 -17786.892,E2 -17786.892} C_VEL
LIN {X 0,Y 270.192,Z 596.81,A -85,B 0,C 180,E1 -17790.382,E2 -17790.382} C_VEL
LIN {X 0,Y 270.259,Z 596.819,A -85,B 0,C 180,E1 -17793.763,E2 -17793.763} C_VEL
LIN {X 0,Y 270.226,Z 596.801,A -85,B 0,C 180,E1 -17797.038,E2 -17797.038} C_VEL
LIN {X 0,Y 270.296,Z 596.815,A -85,B 0,C 180,E1 -17800.244,E2 -17800.244} C_VEL
LIN {X 0,Y 270.39,Z 596.783,A -85,B 0,C 180,E1 -17804.935,E2 -17804.935} C_VEL
LIN {X 0,Y 270.406,Z 596.789,A -85,B 0,C 180,E1 -17809.518,E2 -17809.518} C_VEL
LIN {X 0,Y 270.593,Z 596.761,A -85,B 0,C 180,E1 -17812.538,E2 -17812.538} C_VEL
LIN {X 0,Y 270.782,Z 596.729,A -85,B 0,C 180,E1 -17818.513,E2 -17818.513} C_VEL
LIN {X 0,Y 270.784,Z 596.754,A -85,B 0,C 180,E1 -17821.487,E2 -17821.487} C_VEL
LIN {X 0,Y 270.601,Z 596.767,A -85,B 0,C 180,E1 -17827.461,E2 -17827.461} C_VEL
LIN {X 0,Y 270.435,Z 596.792,A -85,B 0,C 180,E1 -17830.481,E2 -17830.481} C_VEL
LIN {X 0,Y 270.397,Z 596.801,A -85,B 0,C 180,E1 -17835.065,E2 -17835.065} C_VEL
LIN {X 0,Y 270.296,Z 596.8,A -85,B 0,C 180,E1 -17839.756,E2 -17839.756} C_VEL
LIN {X 0,Y 270.269,Z 596.802,A -85,B 0,C 180,E1 -17844.586,E2 -17844.586} C_VEL
LIN {X 0,Y 270.267,Z 596.818,A -85,B 0,C 180,E1 -17847.909,E2 -17847.909} C_VEL
LIN {X 0,Y 270.181,Z 596.825,A -85,B 0,C 180,E1 -17851.349,E2 -17851.349} C_VEL
LIN {X 0,Y 270.211,Z 596.815,A -85,B 0,C 180,E1 -17854.904,E2 -17854.904} C_VEL
LIN {X 0,Y 270.219,Z 596.826,A -85,B 0,C 180,E1 -17858.718,E2 -17858.718} C_VEL
LIN {X 0,Y 270.191,Z 596.793,A -85,B 0,C 180,E1 -17862.555,E2 -17862.555} C_VEL
LIN {X 0,Y 270.207,Z 596.874,A -85,B 0,C 180,E1 -17864.811,E2 -17864.811} C_VEL
LIN {X 0,Y 271.143,Z 599.631,A -85,B 0,C 180,E1 -17865.058,E2 -17865.058} C_VEL
LIN {X 0,Y 272.869,Z 602.003,A -85,B 0,C 180,E1 -17865.419,E2 -17865.419} C_VEL
LIN {X 0,Y 281.652,Z 616.663,A -85,B 0,C 180,E1 -17867.238,E2 -17867.238} C_VEL
LIN {X 0,Y 288.736,Z 629.829,A -85,B 0,C 180,E1 -17868.632,E2 -17868.632} C_VEL
LIN {X 0,Y 291.162,Z 634.709,A -85,B 0,C 180,E1 -17869.099,E2 -17869.099} C_VEL
LIN {X 0,Y 289.255,Z 690.855,A -85,B 0,C 180,E1 -17870.502,E2 -17870.502} C_VEL
LIN {X 0,Y 288.571,Z 704.18,A -85,B 0,C 180,E1 -17871.07,E2 -17871.07} C_VEL
LIN {X 0,Y 287.443,Z 717.248,A -85,B 0,C 180,E1 -17871.921,E2 -17871.921} C_VEL
LIN {X 0,Y 285.86,Z 728.969,A -85,B 0,C 180,E1 -17872.963,E2 -17872.963} C_VEL
LIN {X 0,Y 284.069,Z 739.951,A -85,B 0,C 180,E1 -17874.234,E2 -17874.234} C_VEL
LIN {X 0,Y 282.111,Z 749.979,A -85,B 0,C 180,E1 -17875.693,E2 -17875.693} C_VEL
LIN {X 0,Y 280.001,Z 759.103,A -85,B 0,C 180,E1 -17877.341,E2 -17877.341} C_VEL
LIN {X 0,Y 277.902,Z 767.742,A -85,B 0,C 180,E1 -17879.299,E2 -17879.299} C_VEL
LIN {X 0,Y 275.775,Z 775.405,A -85,B 0,C 180,E1 -17881.457,E2 -17881.457} C_VEL
LIN {X 0,Y 274.091,Z 780.986,A -85,B 0,C 180,E1 -17883.421,E2 -17883.421} C_VEL
LIN {X 0,Y 272.58,Z 785.976,A -85,B 0,C 180,E1 -17885.637,E2 -17885.637} C_VEL
LIN {X 0,Y 271.3,Z 789.916,A -85,B 0,C 180,E1 -17887.938,E2 -17887.938} C_VEL
LIN {X 0,Y 270.327,Z 792.756,A -85,B 0,C 180,E1 -17890.247,E2 -17890.247} C_VEL
LIN {X 0,Y 269.775,Z 794.068,A -85,B 0,C 180,E1 -17891.784,E2 -17891.784} C_VEL
LIN {X 0,Y 269.382,Z 794.974,A -85,B 0,C 180,E1 -17893.323,E2 -17893.323} C_VEL
LIN {X 0,Y 269.099,Z 795.5,A -85,B 0,C 180,E1 -17895.088,E2 -17895.088} C_VEL
LIN {X 0,Y 268.778,Z 795.196,A -85,B 0,C 180,E1 -17897.926,E2 -17897.926} C_VEL
LIN {X 0,Y 268.791,Z 794.469,A -85,B 0,C 180,E1 -17899.454,E2 -17899.454} C_VEL
LIN {X 0,Y 268.893,Z 793.313,A -85,B 0,C 180,E1 -17900.978,E2 -17900.978} C_VEL
LIN {X 0,Y 269.147,Z 791.289,A -85,B 0,C 180,E1 -17902.868,E2 -17902.868} C_VEL
LIN {X 0,Y 269.665,Z 787.284,A -85,B 0,C 180,E1 -17905.516,E2 -17905.516} C_VEL
LIN {X 0,Y 270.239,Z 782.686,A -85,B 0,C 180,E1 -17907.764,E2 -17907.764} C_VEL
LIN {X 0,Y 271.32,Z 775.751,A -85,B 0,C 180,E1 -17910.371,E2 -17910.371} C_VEL
LIN {X 0,Y 272.447,Z 768.218,A -85,B 0,C 180,E1 -17912.587,E2 -17912.587} C_VEL
LIN {X 0,Y 273.987,Z 758.749,A -85,B 0,C 180,E1 -17914.782,E2 -17914.782} C_VEL
LIN {X 0,Y 275.342,Z 749.009,A -85,B 0,C 180,E1 -17916.595,E2 -17916.595} C_VEL
LIN {X 0,Y 276.763,Z 738.022,A -85,B 0,C 180,E1 -17918.212,E2 -17918.212} C_VEL
LIN {X 0,Y 278.017,Z 727.304,A -85,B 0,C 180,E1 -17919.457,E2 -17919.457} C_VEL
LIN {X 0,Y 279.1,Z 715.521,A -85,B 0,C 180,E1 -17920.519,E2 -17920.519} C_VEL
LIN {X 0,Y 279.889,Z 702.416,A -85,B 0,C 180,E1 -17921.37,E2 -17921.37} C_VEL
LIN {X 0,Y 280.369,Z 689.562,A -85,B 0,C 180,E1 -17921.913,E2 -17921.913} C_VEL
LIN {X 0,Y 281.938,Z 624.84,A -85,B 0,C 180,E1 -17923.548,E2 -17923.548} C_VEL
LIN {X 0,Y 273.105,Z 603.538,A -85,B 0,C 180,E1 -17924.889,E2 -17924.889} C_VEL
LIN {X 0,Y 270.536,Z 597.468,A -85,B 0,C 180,E1 -17925.293,E2 -17925.293} C_VEL
LIN {X 0,Y 270.405,Z 596.799,A -85,B 0,C 180,E1 -17925.33,E2 -17925.33} C_VEL
LIN {X 0,Y 270.332,Z 596.911,A -85,B 0,C 180,E1 -17928.227,E2 -17928.227} C_VEL
LIN {X 0,Y 272.028,Z 601.344,A -85,B 0,C 180,E1 -17928.523,E2 -17928.523} C_VEL
LIN {X 0,Y 282.703,Z 626.92,A -85,B 0,C 180,E1 -17930.222,E2 -17930.222} C_VEL
LIN {X 0,Y 280.557,Z 692.322,A -85,B 0,C 180,E1 -17932.094,E2 -17932.094} C_VEL
LIN {X 0,Y 279.986,Z 705.723,A -85,B 0,C 180,E1 -17932.774,E2 -17932.774} C_VEL
LIN {X 0,Y 279.025,Z 718.092,A -85,B 0,C 180,E1 -17933.667,E2 -17933.667} C_VEL
LIN {X 0,Y 277.84,Z 730.036,A -85,B 0,C 180,E1 -17934.832,E2 -17934.832} C_VEL
LIN {X 0,Y 276.624,Z 740.939,A -85,B 0,C 180,E1 -17936.195,E2 -17936.195} C_VEL
LIN {X 0,Y 275.259,Z 751.129,A -85,B 0,C 180,E1 -17937.772,E2 -17937.772} C_VEL
LIN {X 0,Y 273.807,Z 760.873,A -85,B 0,C 180,E1 -17939.646,E2 -17939.646} C_VEL
LIN {X 0,Y 272.369,Z 770.162,A -85,B 0,C 180,E1 -17941.886,E2 -17941.886} C_VEL
LIN {X 0,Y 271.112,Z 778.167,A -85,B 0,C 180,E1 -17944.337,E2 -17944.337} C_VEL
LIN {X 0,Y 270.246,Z 784.259,A -85,B 0,C 180,E1 -17946.736,E2 -17946.736} C_VEL
LIN {X 0,Y 269.66,Z 788.234,A -85,B 0,C 180,E1 -17948.718,E2 -17948.718} C_VEL
LIN {X 0,Y 269.172,Z 791.47,A -85,B 0,C 180,E1 -17950.784,E2 -17950.784} C_VEL
LIN {X 0,Y 268.863,Z 793.943,A -85,B 0,C 180,E1 -17952.953,E2 -17952.953} C_VEL
LIN {X 0,Y 268.734,Z 795.494,A -85,B 0,C 180,E1 -17955.08,E2 -17955.08} C_VEL
LIN {X 0,Y 268.817,Z 796.207,A -85,B 0,C 180,E1 -17957.256,E2 -17957.256} C_VEL
LIN {X 0,Y 269.055,Z 796.161,A -85,B 0,C 180,E1 -17959.243,E2 -17959.243} C_VEL
LIN {X 0,Y 269.576,Z 795.258,A -85,B 0,C 180,E1 -17961.453,E2 -17961.453} C_VEL
LIN {X 0,Y 270.322,Z 793.37,A -85,B 0,C 180,E1 -17963.739,E2 -17963.739} C_VEL
LIN {X 0,Y 270.112,Z 792.063,A -85,B 0,C 180,E1 -17964.956,E2 -17964.956} C_VEL
LIN {X 0,Y 268.205,Z 789.644,A -85,B 0,C 180,E1 -17966.968,E2 -17966.968} C_VEL
LIN {X 0,Y 266.509,Z 786.613,A -85,B 0,C 180,E1 -17968.962,E2 -17968.962} C_VEL
LIN {X 0,Y 266.623,Z 784.243,A -85,B 0,C 180,E1 -17970.127,E2 -17970.127} C_VEL
LIN {X 0,Y 268.766,Z 777.275,A -85,B 0,C 180,E1 -17972.754,E2 -17972.754} C_VEL
LIN {X 0,Y 270.805,Z 769.871,A -85,B 0,C 180,E1 -17974.911,E2 -17974.911} C_VEL
LIN {X 0,Y 273.282,Z 760.335,A -85,B 0,C 180,E1 -17977.109,E2 -17977.109} C_VEL
LIN {X 0,Y 275.531,Z 750.624,A -85,B 0,C 180,E1 -17978.882,E2 -17978.882} C_VEL
LIN {X 0,Y 277.74,Z 739.237,A -85,B 0,C 180,E1 -17980.529,E2 -17980.529} C_VEL
LIN {X 0,Y 279.509,Z 728.434,A -85,B 0,C 180,E1 -17981.757,E2 -17981.757} C_VEL
LIN {X 0,Y 281.092,Z 716.173,A -85,B 0,C 180,E1 -17982.822,E2 -17982.822} C_VEL
LIN {X 0,Y 282.196,Z 702.683,A -85,B 0,C 180,E1 -17983.683,E2 -17983.683} C_VEL
LIN {X 0,Y 282.891,Z 689.955,A -85,B 0,C 180,E1 -17984.195,E2 -17984.195} C_VEL
LIN {X 0,Y 285.468,Z 636.207,A -85,B 0,C 180,E1 -17985.796,E2 -17985.796} C_VEL
LIN {X 0,Y 279.749,Z 624.751,A -85,B 0,C 180,E1 -17987.183,E2 -17987.183} C_VEL
LIN {X 0,Y 273.783,Z 614.362,A -85,B 0,C 180,E1 -17988.689,E2 -17988.689} C_VEL
LIN {X 0,Y 268.27,Z 605.92,A -85,B 0,C 180,E1 -17990.148,E2 -17990.148} C_VEL
LIN {X 0,Y 265.903,Z 602.12,A -85,B 0,C 180,E1 -17990.827,E2 -17990.827} C_VEL
LIN {X 0,Y 264.125,Z 599.792,A -85,B 0,C 180,E1 -17991.333,E2 -17991.333} C_VEL
LIN {X 0,Y 263.532,Z 597.66,A -85,B 0,C 180,E1 -17991.614,E2 -17991.614} C_VEL
LIN {X 0,Y 263.51,Z 597.663,A -85,B 0,C 180,E1 -17993.876,E2 -17993.876} C_VEL
LIN {X 0,Y 263.746,Z 597.629,A -85,B 0,C 180,E1 -17998.473,E2 -17998.473} C_VEL
LIN {X 0,Y 263.746,Z 597.631,A -85,B 0,C 180,E1 -18001.527,E2 -18001.527} C_VEL
LIN {X 0,Y 263.565,Z 597.647,A -85,B 0,C 180,E1 -18007.662,E2 -18007.662} C_VEL
LIN {X 0,Y 263.368,Z 597.667,A -85,B 0,C 180,E1 -18010.766,E2 -18010.766} C_VEL
LIN {X 0,Y 263.339,Z 597.675,A -85,B 0,C 180,E1 -18015.479,E2 -18015.479} C_VEL
LIN {X 0,Y 263.258,Z 597.68,A -85,B 0,C 180,E1 -18020.307,E2 -18020.307} C_VEL
LIN {X 0,Y 263.204,Z 597.698,A -85,B 0,C 180,E1 -18025.292,E2 -18025.292} C_VEL
LIN {X 0,Y 263.175,Z 597.702,A -85,B 0,C 180,E1 -18028.73,E2 -18028.73} C_VEL
LIN {X 0,Y 263.129,Z 597.71,A -85,B 0,C 180,E1 -18032.289,E2 -18032.289} C_VEL
LIN {X 0,Y 263.186,Z 597.698,A -85,B 0,C 180,E1 -18035.978,E2 -18035.978} C_VEL
LIN {X 0,Y 263.157,Z 597.702,A -85,B 0,C 180,E1 -18039.863,E2 -18039.863} C_VEL
LIN {X 0,Y 263.143,Z 597.705,A -85,B 0,C 180,E1 -18043.98,E2 -18043.98} C_VEL
LIN {X 0,Y 263.189,Z 597.904,A -85,B 0,C 180,E1 -18044.504,E2 -18044.504} C_VEL
LIN {X 0,Y 265.753,Z 605.99,A -85,B 0,C 180,E1 -18048.614,E2 -18048.614} C_VEL
LIN {X 0,Y 267.805,Z 613.531,A -85,B 0,C 180,E1 -18051.933,E2 -18051.933} C_VEL
LIN {X 0,Y 269.634,Z 621.276,A -85,B 0,C 180,E1 -18055.011,E2 -18055.011} C_VEL
LIN {X 0,Y 270.079,Z 623.143,A -85,B 0,C 180,E1 -18055.633,E2 -18055.633} C_VEL
LIN {X 0,Y 272.516,Z 628.063,A -85,B 0,C 180,E1 -18056.312,E2 -18056.312} C_VEL
LIN {X 0,Y 277.594,Z 639.569,A -85,B 0,C 180,E1 -18057.697,E2 -18057.697} C_VEL
LIN {X 0,Y 280.714,Z 659.017,A -85,B 0,C 180,E1 -18058.977,E2 -18058.977} C_VEL
LIN {X 0,Y 282.415,Z 674.115,A -85,B 0,C 180,E1 -18059.816,E2 -18059.816} C_VEL
LIN {X 0,Y 283.499,Z 688.461,A -85,B 0,C 180,E1 -18060.505,E2 -18060.505} C_VEL
LIN {X 0,Y 281.094,Z 736.224,A -85,B 0,C 180,E1 -18061.943,E2 -18061.943} C_VEL
LIN {X 0,Y 279.755,Z 749.65,A -85,B 0,C 180,E1 -18062.611,E2 -18062.611} C_VEL
LIN {X 0,Y 277.999,Z 761.539,A -85,B 0,C 180,E1 -18063.44,E2 -18063.44} C_VEL
LIN {X 0,Y 275.848,Z 773.27,A -85,B 0,C 180,E1 -18064.537,E2 -18064.537} C_VEL
LIN {X 0,Y 273.401,Z 784.697,A -85,B 0,C 180,E1 -18065.916,E2 -18065.916} C_VEL
LIN {X 0,Y 271.01,Z 795.157,A -85,B 0,C 180,E1 -18067.512,E2 -18067.512} C_VEL
LIN {X 0,Y 268.645,Z 804.648,A -85,B 0,C 180,E1 -18069.319,E2 -18069.319} C_VEL
LIN {X 0,Y 266.393,Z 813.929,A -85,B 0,C 180,E1 -18071.544,E2 -18071.544} C_VEL
LIN {X 0,Y 264.585,Z 821.487,A -85,B 0,C 180,E1 -18073.806,E2 -18073.806} C_VEL
LIN {X 0,Y 263.132,Z 827.6,A -85,B 0,C 180,E1 -18076.091,E2 -18076.091} C_VEL
LIN {X 0,Y 262.105,Z 832.483,A -85,B 0,C 180,E1 -18078.399,E2 -18078.399} C_VEL
LIN {X 0,Y 261.612,Z 836.291,A -85,B 0,C 180,E1 -18080.725,E2 -18080.725} C_VEL
LIN {X 0,Y 261.459,Z 838.246,A -85,B 0,C 180,E1 -18082.276,E2 -18082.276} C_VEL
LIN {X 0,Y 261.454,Z 839.949,A -85,B 0,C 180,E1 -18084.031,E2 -18084.031} C_VEL
LIN {X 0,Y 261.569,Z 841.61,A -85,B 0,C 180,E1 -18086.92,E2 -18086.92} C_VEL
LIN {X 0,Y 261.84,Z 841.882,A -85,B 0,C 180,E1 -18088.462,E2 -18088.462} C_VEL
LIN {X 0,Y 261.927,Z 841.72,A -85,B 0,C 180,E1 -18090,E2 -18090} C_VEL
LIN {X 0,Y 261.68,Z 840.403,A -85,B 0,C 180,E1 -18093.079,E2 -18093.079} C_VEL
LIN {X 0,Y 261.474,Z 839.025,A -85,B 0,C 180,E1 -18096.011,E2 -18096.011} C_VEL
LIN {X 0,Y 261.433,Z 837.527,A -85,B 0,C 180,E1 -18097.724,E2 -18097.724} C_VEL
LIN {X 0,Y 261.728,Z 834.685,A -85,B 0,C 180,E1 -18100.052,E2 -18100.052} C_VEL
LIN {X 0,Y 262.373,Z 830.83,A -85,B 0,C 180,E1 -18102.374,E2 -18102.374} C_VEL
LIN {X 0,Y 263.602,Z 825.871,A -85,B 0,C 180,E1 -18104.672,E2 -18104.672} C_VEL
LIN {X 0,Y 265.187,Z 819.652,A -85,B 0,C 180,E1 -18106.949,E2 -18106.949} C_VEL
LIN {X 0,Y 267.009,Z 811.946,A -85,B 0,C 180,E1 -18109.208,E2 -18109.208} C_VEL
LIN {X 0,Y 269.599,Z 802.316,A -85,B 0,C 180,E1 -18111.404,E2 -18111.404} C_VEL
LIN {X 0,Y 272.153,Z 792.401,A -85,B 0,C 180,E1 -18113.191,E2 -18113.191} C_VEL
LIN {X 0,Y 274.665,Z 781.214,A -85,B 0,C 180,E1 -18114.771,E2 -18114.771} C_VEL
LIN {X 0,Y 276.845,Z 770.283,A -85,B 0,C 180,E1 -18115.97,E2 -18115.97} C_VEL
LIN {X 0,Y 278.836,Z 758.194,A -85,B 0,C 180,E1 -18116.98,E2 -18116.98} C_VEL
LIN {X 0,Y 280.564,Z 744.598,A -85,B 0,C 180,E1 -18117.759,E2 -18117.759} C_VEL
LIN {X 0,Y 281.386,Z 732.298,A -85,B 0,C 180,E1 -18118.228,E2 -18118.228} C_VEL
LIN {X 0,Y 283.127,Z 684.441,A -85,B 0,C 180,E1 -18119.446,E2 -18119.446} C_VEL
LIN {X 0,Y 280.647,Z 658.043,A -85,B 0,C 180,E1 -18120.589,E2 -18120.589} C_VEL
LIN {X 0,Y 277.671,Z 635.885,A -85,B 0,C 180,E1 -18121.708,E2 -18121.708} C_VEL
LIN {X 0,Y 270.133,Z 617.611,A -85,B 0,C 180,E1 -18123.471,E2 -18123.471} C_VEL
LIN {X 0,Y 268.551,Z 613.717,A -85,B 0,C 180,E1 -18123.934,E2 -18123.934} C_VEL
LIN {X 0,Y 265.747,Z 606.189,A -85,B 0,C 180,E1 -18124.992,E2 -18124.992} C_VEL
LIN {X 0,Y 263.978,Z 601.132,A -85,B 0,C 180,E1 -18125.755,E2 -18125.755} C_VEL
LIN {X 0,Y 263.199,Z 597.701,A -85,B 0,C 180,E1 -18126.768,E2 -18126.768} C_VEL
LIN {X 0,Y 263.153,Z 597.706,A -85,B 0,C 180,E1 -18129.863,E2 -18129.863} C_VEL
LIN {X 0,Y 263.141,Z 597.708,A -85,B 0,C 180,E1 -18133.979,E2 -18133.979} C_VEL
LIN {X 0,Y 263.171,Z 597.702,A -85,B 0,C 180,E1 -18138.394,E2 -18138.394} C_VEL
LIN {X 0,Y 263.186,Z 597.698,A -85,B 0,C 180,E1 -18142.107,E2 -18142.107} C_VEL
LIN {X 0,Y 263.18,Z 597.684,A -85,B 0,C 180,E1 -18145.89,E2 -18145.89} C_VEL
LIN {X 0,Y 263.137,Z 597.699,A -85,B 0,C 180,E1 -18149.505,E2 -18149.505} C_VEL
LIN {X 0,Y 263.188,Z 597.696,A -85,B 0,C 180,E1 -18153.002,E2 -18153.002} C_VEL
LIN {X 0,Y 263.178,Z 597.683,A -85,B 0,C 180,E1 -18156.386,E2 -18156.386} C_VEL
LIN {X 0,Y 263.258,Z 597.689,A -85,B 0,C 180,E1 -18159.693,E2 -18159.693} C_VEL
LIN {X 0,Y 263.339,Z 597.658,A -85,B 0,C 180,E1 -18164.521,E2 -18164.521} C_VEL
LIN {X 0,Y 263.349,Z 597.672,A -85,B 0,C 180,E1 -18169.233,E2 -18169.233} C_VEL
LIN {X 0,Y 263.553,Z 597.636,A -85,B 0,C 180,E1 -18172.338,E2 -18172.338} C_VEL
LIN {X 0,Y 263.746,Z 597.605,A -85,B 0,C 180,E1 -18178.473,E2 -18178.473} C_VEL
LIN {X 0,Y 263.748,Z 597.631,A -85,B 0,C 180,E1 -18181.527,E2 -18181.527} C_VEL
LIN {X 0,Y 263.563,Z 597.646,A -85,B 0,C 180,E1 -18187.662,E2 -18187.662} C_VEL
LIN {X 0,Y 263.367,Z 597.668,A -85,B 0,C 180,E1 -18190.766,E2 -18190.766} C_VEL
LIN {X 0,Y 263.345,Z 597.682,A -85,B 0,C 180,E1 -18195.478,E2 -18195.478} C_VEL
LIN {X 0,Y 263.258,Z 597.682,A -85,B 0,C 180,E1 -18200.307,E2 -18200.307} C_VEL
LIN {X 0,Y 263.204,Z 597.684,A -85,B 0,C 180,E1 -18205.292,E2 -18205.292} C_VEL
LIN {X 0,Y 263.175,Z 597.694,A -85,B 0,C 180,E1 -18208.73,E2 -18208.73} C_VEL
LIN {X 0,Y 263.13,Z 597.709,A -85,B 0,C 180,E1 -18212.289,E2 -18212.289} C_VEL
LIN {X 0,Y 263.185,Z 597.702,A -85,B 0,C 180,E1 -18215.979,E2 -18215.979} C_VEL
LIN {X 0,Y 263.137,Z 597.697,A -85,B 0,C 180,E1 -18219.867,E2 -18219.867} C_VEL
LIN {X 0,Y 263.146,Z 597.818,A -85,B 0,C 180,E1 -18223.619,E2 -18223.619} C_VEL
LIN {X 0,Y 264.175,Z 600.633,A -85,B 0,C 180,E1 -18223.901,E2 -18223.901} C_VEL
LIN {X 0,Y 265.927,Z 603.004,A -85,B 0,C 180,E1 -18224.289,E2 -18224.289} C_VEL
LIN {X 0,Y 274.745,Z 617.319,A -85,B 0,C 180,E1 -18226.215,E2 -18226.215} C_VEL
LIN {X 0,Y 282.829,Z 632.231,A -85,B 0,C 180,E1 -18227.885,E2 -18227.885} C_VEL
LIN {X 0,Y 285.219,Z 636.952,A -85,B 0,C 180,E1 -18228.363,E2 -18228.363} C_VEL
LIN {X 0,Y 283.281,Z 690.765,A -85,B 0,C 180,E1 -18229.723,E2 -18229.723} C_VEL
LIN {X 0,Y 282.593,Z 704.092,A -85,B 0,C 180,E1 -18230.288,E2 -18230.288} C_VEL
LIN {X 0,Y 281.425,Z 717.338,A -85,B 0,C 180,E1 -18231.152,E2 -18231.152} C_VEL
LIN {X 0,Y 279.745,Z 729.439,A -85,B 0,C 180,E1 -18232.24,E2 -18232.24} C_VEL
LIN {X 0,Y 277.875,Z 740.439,A -85,B 0,C 180,E1 -18233.534,E2 -18233.534} C_VEL
LIN {X 0,Y 275.727,Z 750.929,A -85,B 0,C 180,E1 -18235.093,E2 -18235.093} C_VEL
LIN {X 0,Y 273.395,Z 760.524,A -85,B 0,C 180,E1 -18236.89,E2 -18236.89} C_VEL
LIN {X 0,Y 271.302,Z 768.663,A -85,B 0,C 180,E1 -18238.796,E2 -18238.796} C_VEL
LIN {X 0,Y 268.98,Z 776.56,A -85,B 0,C 180,E1 -18241.095,E2 -18241.095} C_VEL
LIN {X 0,Y 266.915,Z 783.043,A -85,B 0,C 180,E1 -18243.539,E2 -18243.539} C_VEL
LIN {X 0,Y 265.432,Z 787.623,A -85,B 0,C 180,E1 -18245.771,E2 -18245.771} C_VEL
LIN {X 0,Y 264.161,Z 791.285,A -85,B 0,C 180,E1 -18248.133,E2 -18248.133} C_VEL
LIN {X 0,Y 263.476,Z 793.143,A -85,B 0,C 180,E1 -18249.711,E2 -18249.711} C_VEL
LIN {X 0,Y 262.858,Z 794.531,A -85,B 0,C 180,E1 -18251.287,E2 -18251.287} C_VEL
LIN {X 0,Y 262.135,Z 796.029,A -85,B 0,C 180,E1 -18254.449,E2 -18254.449} C_VEL
LIN {X 0,Y 261.904,Z 796.165,A -85,B 0,C 180,E1 -18256.025,E2 -18256.025} C_VEL
LIN {X 0,Y 261.708,Z 795.187,A -85,B 0,C 180,E1 -18259.165,E2 -18259.165} C_VEL
LIN {X 0,Y 261.796,Z 794.109,A -85,B 0,C 180,E1 -18260.731,E2 -18260.731} C_VEL
LIN {X 0,Y 262.076,Z 791.932,A -85,B 0,C 180,E1 -18262.848,E2 -18262.848} C_VEL
LIN {X 0,Y 262.547,Z 788.257,A -85,B 0,C 180,E1 -18265.394,E2 -18265.394} C_VEL
LIN {X 0,Y 263.151,Z 783.763,A -85,B 0,C 180,E1 -18267.704,E2 -18267.704} C_VEL
LIN {X 0,Y 264.209,Z 776.942,A -85,B 0,C 180,E1 -18270.381,E2 -18270.381} C_VEL
LIN {X 0,Y 265.381,Z 769.57,A -85,B 0,C 180,E1 -18272.656,E2 -18272.656} C_VEL
LIN {X 0,Y 266.648,Z 762.008,A -85,B 0,C 180,E1 -18274.535,E2 -18274.535} C_VEL
LIN {X 0,Y 268.187,Z 751.773,A -85,B 0,C 180,E1 -18276.583,E2 -18276.583} C_VEL
LIN {X 0,Y 269.601,Z 741.413,A -85,B 0,C 180,E1 -18278.243,E2 -18278.243} C_VEL
LIN {X 0,Y 271.084,Z 729.699,A -85,B 0,C 180,E1 -18279.701,E2 -18279.701} C_VEL
LIN {X 0,Y 272.282,Z 717.833,A -85,B 0,C 180,E1 -18280.837,E2 -18280.837} C_VEL
LIN {X 0,Y 273.036,Z 705.712,A -85,B 0,C 180,E1 -18281.707,E2 -18281.707} C_VEL
LIN {X 0,Y 273.605,Z 692.842,A -85,B 0,C 180,E1 -18282.316,E2 -18282.316} C_VEL
LIN {X 0,Y 275.307,Z 626.478,A -85,B 0,C 180,E1 -18284.055,E2 -18284.055} C_VEL
LIN {X 0,Y 266.621,Z 605.483,A -85,B 0,C 180,E1 -18285.425,E2 -18285.425} C_VEL
LIN {X 0,Y 263.51,Z 598.453,A -85,B 0,C 180,E1 -18285.926,E2 -18285.926} C_VEL
LIN {X 0,Y 263.349,Z 597.677,A -85,B 0,C 180,E1 -18286.008,E2 -18286.008} C_VEL
LIN {X 0,Y 263.268,Z 597.692,A -85,B 0,C 180,E1 -18287.576,E2 -18287.576} C_VEL
LIN {X 0,Y 264.886,Z 602.06,A -85,B 0,C 180,E1 -18287.902,E2 -18287.902} C_VEL
LIN {X 0,Y 275.155,Z 626.337,A -85,B 0,C 180,E1 -18289.599,E2 -18289.599} C_VEL
LIN {X 0,Y 276.078,Z 629.025,A -85,B 0,C 180,E1 -18289.76,E2 -18289.76} C_VEL
LIN {X 0,Y 273.85,Z 692.486,A -85,B 0,C 180,E1 -18291.615,E2 -18291.615} C_VEL
LIN {X 0,Y 273.274,Z 706.064,A -85,B 0,C 180,E1 -18292.316,E2 -18292.316} C_VEL
LIN {X 0,Y 272.209,Z 719.171,A -85,B 0,C 180,E1 -18293.287,E2 -18293.287} C_VEL
LIN {X 0,Y 270.946,Z 731.344,A -85,B 0,C 180,E1 -18294.52,E2 -18294.52} C_VEL
LIN {X 0,Y 269.528,Z 743.5,A -85,B 0,C 180,E1 -18296.112,E2 -18296.112} C_VEL
LIN {X 0,Y 267.957,Z 754.253,A -85,B 0,C 180,E1 -18297.908,E2 -18297.908} C_VEL
LIN {X 0,Y 266.617,Z 763.27,A -85,B 0,C 180,E1 -18299.775,E2 -18299.775} C_VEL
LIN {X 0,Y 265.207,Z 771.993,A -85,B 0,C 180,E1 -18302.005,E2 -18302.005} C_VEL
LIN {X 0,Y 263.996,Z 779.342,A -85,B 0,C 180,E1 -18304.384,E2 -18304.384} C_VEL
LIN {X 0,Y 263.141,Z 785.126,A -85,B 0,C 180,E1 -18306.751,E2 -18306.751} C_VEL
LIN {X 0,Y 262.506,Z 789.526,A -85,B 0,C 180,E1 -18309.067,E2 -18309.067} C_VEL
LIN {X 0,Y 261.851,Z 793.692,A -85,B 0,C 180,E1 -18312.142,E2 -18312.142} C_VEL
LIN {X 0,Y 261.67,Z 795.582,A -85,B 0,C 180,E1 -18314.29,E2 -18314.29} C_VEL
LIN {X 0,Y 261.689,Z 796.666,A -85,B 0,C 180,E1 -18316.477,E2 -18316.477} C_VEL
LIN {X 0,Y 261.895,Z 796.916,A -85,B 0,C 180,E1 -18318.709,E2 -18318.709} C_VEL
LIN {X 0,Y 262.382,Z 796.308,A -85,B 0,C 180,E1 -18320.965,E2 -18320.965} C_VEL
LIN {X 0,Y 263.396,Z 794.069,A -85,B 0,C 180,E1 -18324.055,E2 -18324.055} C_VEL
LIN {X 0,Y 264.715,Z 790.228,A -85,B 0,C 180,E1 -18327.027,E2 -18327.027} C_VEL
LIN {X 0,Y 266.487,Z 784.7,A -85,B 0,C 180,E1 -18329.928,E2 -18329.928} C_VEL
LIN {X 0,Y 266.623,Z 784.243,A -85,B 0,C 180,E1 -18330.127,E2 -18330.127} C_VEL
LIN {X 0,Y 266.8,Z 781.664,A -85,B 0,C 180,E1 -18331.269,E2 -18331.269} C_VEL
LIN {X 0,Y 265.52,Z 777.268,A -85,B 0,C 180,E1 -18333.168,E2 -18333.168} C_VEL
LIN {X 0,Y 264.452,Z 772.332,A -85,B 0,C 180,E1 -18335.005,E2 -18335.005} C_VEL
LIN {X 0,Y 264.932,Z 768.79,A -85,B 0,C 180,E1 -18336.025,E2 -18336.025} C_VEL
LIN {X 0,Y 267.152,Z 760.552,A -85,B 0,C 180,E1 -18337.914,E2 -18337.914} C_VEL
LIN {X 0,Y 269.62,Z 750.312,A -85,B 0,C 180,E1 -18339.778,E2 -18339.778} C_VEL
LIN {X 0,Y 271.765,Z 739.627,A -85,B 0,C 180,E1 -18341.336,E2 -18341.336} C_VEL
LIN {X 0,Y 273.729,Z 728.027,A -85,B 0,C 180,E1 -18342.657,E2 -18342.657} C_VEL
LIN {X 0,Y 275.442,Z 714.808,A -85,B 0,C 180,E1 -18343.787,E2 -18343.787} C_VEL
LIN {X 0,Y 276.511,Z 702.136,A -85,B 0,C 180,E1 -18344.579,E2 -18344.579} C_VEL
LIN {X 0,Y 277.285,Z 687.631,A -85,B 0,C 180,E1 -18345.134,E2 -18345.134} C_VEL
LIN {X 0,Y 279.906,Z 638.842,A -85,B 0,C 180,E1 -18346.598,E2 -18346.598} C_VEL
LIN {X 0,Y 274.024,Z 627.098,A -85,B 0,C 180,E1 -18348.104,E2 -18348.104} C_VEL
LIN {X 0,Y 268.336,Z 617.445,A -85,B 0,C 180,E1 -18349.627,E2 -18349.627} C_VEL
LIN {X 0,Y 263.778,Z 610.336,A -85,B 0,C 180,E1 -18350.916,E2 -18350.916} C_VEL
LIN {X 0,Y 261.699,Z 607.083,A -85,B 0,C 180,E1 -18351.541,E2 -18351.541} C_VEL
LIN {X 0,Y 259.662,Z 603.749,A -85,B 0,C 180,E1 -18352.178,E2 -18352.178} C_VEL
LIN {X 0,Y 257.294,Z 601.026,A -85,B 0,C 180,E1 -18352.89,E2 -18352.89} C_VEL
LIN {X 0,Y 256.481,Z 598.536,A -85,B 0,C 180,E1 -18353.263,E2 -18353.263} C_VEL
LIN {X 0,Y 256.709,Z 598.505,A -85,B 0,C 180,E1 -18358.431,E2 -18358.431} C_VEL
LIN {X 0,Y 256.709,Z 598.507,A -85,B 0,C 180,E1 -18361.569,E2 -18361.569} C_VEL
LIN {X 0,Y 256.533,Z 598.524,A -85,B 0,C 180,E1 -18367.873,E2 -18367.873} C_VEL
LIN {X 0,Y 256.304,Z 598.548,A -85,B 0,C 180,E1 -18371.066,E2 -18371.066} C_VEL
LIN {X 0,Y 256.274,Z 598.553,A -85,B 0,C 180,E1 -18375.917,E2 -18375.917} C_VEL
LIN {X 0,Y 256.162,Z 598.564,A -85,B 0,C 180,E1 -18380.896,E2 -18380.896} C_VEL
LIN {X 0,Y 256.184,Z 598.57,A -85,B 0,C 180,E1 -18385.139,E2 -18385.139} C_VEL
LIN {X 0,Y 256.11,Z 598.582,A -85,B 0,C 180,E1 -18389.6,E2 -18389.6} C_VEL
LIN {X 0,Y 256.081,Z 598.581,A -85,B 0,C 180,E1 -18393.291,E2 -18393.291} C_VEL
LIN {X 0,Y 256.138,Z 598.576,A -85,B 0,C 180,E1 -18397.279,E2 -18397.279} C_VEL
LIN {X 0,Y 256.101,Z 598.581,A -85,B 0,C 180,E1 -18401.195,E2 -18401.195} C_VEL
LIN {X 0,Y 256.09,Z 598.706,A -85,B 0,C 180,E1 -18402.847,E2 -18402.847} C_VEL
LIN {X 0,Y 258.283,Z 605.539,A -85,B 0,C 180,E1 -18406.674,E2 -18406.674} C_VEL
LIN {X 0,Y 260.058,Z 611.426,A -85,B 0,C 180,E1 -18409.566,E2 -18409.566} C_VEL
LIN {X 0,Y 262.361,Z 620.43,A -85,B 0,C 180,E1 -18413.478,E2 -18413.478} C_VEL
LIN {X 0,Y 262.713,Z 621.952,A -85,B 0,C 180,E1 -18414.047,E2 -18414.047} C_VEL
LIN {X 0,Y 265.199,Z 626.947,A -85,B 0,C 180,E1 -18414.809,E2 -18414.809} C_VEL
LIN {X 0,Y 270.429,Z 637.85,A -85,B 0,C 180,E1 -18416.329,E2 -18416.329} C_VEL
LIN {X 0,Y 272.482,Z 643.033,A -85,B 0,C 180,E1 -18416.934,E2 -18416.934} C_VEL
LIN {X 0,Y 275.294,Z 661.549,A -85,B 0,C 180,E1 -18418.175,E2 -18418.175} C_VEL
LIN {X 0,Y 276.862,Z 676.404,A -85,B 0,C 180,E1 -18419.022,E2 -18419.022} C_VEL
LIN {X 0,Y 277.768,Z 688.963,A -85,B 0,C 180,E1 -18419.657,E2 -18419.657} C_VEL
LIN {X 0,Y 275.291,Z 735.428,A -85,B 0,C 180,E1 -18421.089,E2 -18421.089} C_VEL
LIN {X 0,Y 273.865,Z 748.881,A -85,B 0,C 180,E1 -18421.762,E2 -18421.762} C_VEL
LIN {X 0,Y 272.069,Z 760.781,A -85,B 0,C 180,E1 -18422.606,E2 -18422.606} C_VEL
LIN {X 0,Y 269.827,Z 772.527,A -85,B 0,C 180,E1 -18423.719,E2 -18423.719} C_VEL
LIN {X 0,Y 267.267,Z 783.969,A -85,B 0,C 180,E1 -18425.12,E2 -18425.12} C_VEL
LIN {X 0,Y 264.753,Z 794.399,A -85,B 0,C 180,E1 -18426.743,E2 -18426.743} C_VEL
LIN {X 0,Y 261.998,Z 804.706,A -85,B 0,C 180,E1 -18428.769,E2 -18428.769} C_VEL
LIN {X 0,Y 259.632,Z 813.852,A -85,B 0,C 180,E1 -18431.045,E2 -18431.045} C_VEL
LIN {X 0,Y 257.773,Z 821.306,A -85,B 0,C 180,E1 -18433.365,E2 -18433.365} C_VEL
LIN {X 0,Y 256.213,Z 827.312,A -85,B 0,C 180,E1 -18435.708,E2 -18435.708} C_VEL
LIN {X 0,Y 255.09,Z 832.112,A -85,B 0,C 180,E1 -18438.075,E2 -18438.075} C_VEL
LIN {X 0,Y 254.558,Z 835.845,A -85,B 0,C 180,E1 -18440.465,E2 -18440.465} C_VEL
LIN {X 0,Y 254.372,Z 839.247,A -85,B 0,C 180,E1 -18443.655,E2 -18443.655} C_VEL
LIN {X 0,Y 254.413,Z 840.341,A -85,B 0,C 180,E1 -18445.246,E2 -18445.246} C_VEL
LIN {X 0,Y 254.484,Z 841,A -85,B 0,C 180,E1 -18446.834,E2 -18446.834} C_VEL
LIN {X 0,Y 254.775,Z 841.236,A -85,B 0,C 180,E1 -18448.419,E2 -18448.419} C_VEL
LIN {X 0,Y 254.87,Z 841.046,A -85,B 0,C 180,E1 -18450,E2 -18450} C_VEL
LIN {X 0,Y 254.584,Z 839.808,A -85,B 0,C 180,E1 -18453.165,E2 -18453.165} C_VEL
LIN {X 0,Y 254.393,Z 838.635,A -85,B 0,C 180,E1 -18455.98,E2 -18455.98} C_VEL
LIN {X 0,Y 254.357,Z 837.025,A -85,B 0,C 180,E1 -18457.941,E2 -18457.941} C_VEL
LIN {X 0,Y 254.695,Z 834.233,A -85,B 0,C 180,E1 -18460.332,E2 -18460.332} C_VEL
LIN {X 0,Y 255.399,Z 830.434,A -85,B 0,C 180,E1 -18462.717,E2 -18462.717} C_VEL
LIN {X 0,Y 256.68,Z 825.533,A -85,B 0,C 180,E1 -18465.076,E2 -18465.076} C_VEL
LIN {X 0,Y 258.359,Z 819.379,A -85,B 0,C 180,E1 -18467.411,E2 -18467.411} C_VEL
LIN {X 0,Y 260.305,Z 811.766,A -85,B 0,C 180,E1 -18469.723,E2 -18469.723} C_VEL
LIN {X 0,Y 262.528,Z 804.018,A -85,B 0,C 180,E1 -18471.598,E2 -18471.598} C_VEL
LIN {X 0,Y 265.05,Z 794.574,A -85,B 0,C 180,E1 -18473.436,E2 -18473.436} C_VEL
LIN {X 0,Y 267.609,Z 784.129,A -85,B 0,C 180,E1 -18475.054,E2 -18475.054} C_VEL
LIN {X 0,Y 270.141,Z 772.507,A -85,B 0,C 180,E1 -18476.456,E2 -18476.456} C_VEL
LIN {X 0,Y 272.397,Z 760.102,A -85,B 0,C 180,E1 -18477.567,E2 -18477.567} C_VEL
LIN {X 0,Y 274.241,Z 747.073,A -85,B 0,C 180,E1 -18478.404,E2 -18478.404} C_VEL
LIN {X 0,Y 275.34,Z 733.89,A -85,B 0,C 180,E1 -18478.958,E2 -18478.958} C_VEL
LIN {X 0,Y 277.147,Z 684.674,A -85,B 0,C 180,E1 -18480.258,E2 -18480.258} C_VEL
LIN {X 0,Y 274.869,Z 659.498,A -85,B 0,C 180,E1 -18481.377,E2 -18481.377} C_VEL
LIN {X 0,Y 272.049,Z 638.406,A -85,B 0,C 180,E1 -18482.483,E2 -18482.483} C_VEL
LIN {X 0,Y 264.144,Z 618.987,A -85,B 0,C 180,E1 -18484.431,E2 -18484.431} C_VEL
LIN {X 0,Y 261.788,Z 613.264,A -85,B 0,C 180,E1 -18485.115,E2 -18485.115} C_VEL
LIN {X 0,Y 257.546,Z 602.347,A -85,B 0,C 180,E1 -18486.805,E2 -18486.805} C_VEL
LIN {X 0,Y 256.212,Z 599.063,A -85,B 0,C 180,E1 -18487.357,E2 -18487.357} C_VEL
LIN {X 0,Y 256.151,Z 598.573,A -85,B 0,C 180,E1 -18487.511,E2 -18487.511} C_VEL
LIN {X 0,Y 256.083,Z 598.579,A -85,B 0,C 180,E1 -18491.197,E2 -18491.197} C_VEL
LIN {X 0,Y 256.075,Z 598.576,A -85,B 0,C 180,E1 -18495.525,E2 -18495.525} C_VEL
LIN {X 0,Y 256.101,Z 598.581,A -85,B 0,C 180,E1 -18498.805,E2 -18498.805} C_VEL
LIN {X 0,Y 256.152,Z 598.577,A -85,B 0,C 180,E1 -18502.871,E2 -18502.871} C_VEL
LIN {X 0,Y 256.082,Z 598.575,A -85,B 0,C 180,E1 -18506.709,E2 -18506.709} C_VEL
LIN {X 0,Y 256.123,Z 598.56,A -85,B 0,C 180,E1 -18511.409,E2 -18511.409} C_VEL
LIN {X 0,Y 256.162,Z 598.565,A -85,B 0,C 180,E1 -18515.699,E2 -18515.699} C_VEL
LIN {X 0,Y 256.161,Z 598.566,A -85,B 0,C 180,E1 -18519.104,E2 -18519.104} C_VEL
LIN {X 0,Y 256.274,Z 598.537,A -85,B 0,C 180,E1 -18524.083,E2 -18524.083} C_VEL
LIN {X 0,Y 256.287,Z 598.56,A -85,B 0,C 180,E1 -18527.327,E2 -18527.327} C_VEL
LIN {X 0,Y 256.51,Z 598.51,A -85,B 0,C 180,E1 -18532.126,E2 -18532.126} C_VEL
LIN {X 0,Y 256.495,Z 598.519,A -85,B 0,C 180,E1 -18536.859,E2 -18536.859} C_VEL
LIN {X 0,Y 256.76,Z 598.487,A -85,B 0,C 180,E1 -18540,E2 -18540} C_VEL
LIN {X 0,Y 256.498,Z 598.53,A -85,B 0,C 180,E1 -18543.141,E2 -18543.141} C_VEL
LIN {X 0,Y 256.532,Z 598.525,A -85,B 0,C 180,E1 -18547.873,E2 -18547.873} C_VEL
LIN {X 0,Y 256.303,Z 598.545,A -85,B 0,C 180,E1 -18551.066,E2 -18551.066} C_VEL
LIN {X 0,Y 256.294,Z 598.56,A -85,B 0,C 180,E1 -18555.915,E2 -18555.915} C_VEL
LIN {X 0,Y 256.161,Z 598.571,A -85,B 0,C 180,E1 -18560.896,E2 -18560.896} C_VEL
LIN {X 0,Y 256.184,Z 598.557,A -85,B 0,C 180,E1 -18565.139,E2 -18565.139} C_VEL
LIN {X 0,Y 256.11,Z 598.568,A -85,B 0,C 180,E1 -18569.6,E2 -18569.6} C_VEL
LIN {X 0,Y 256.082,Z 598.579,A -85,B 0,C 180,E1 -18573.291,E2 -18573.291} C_VEL
LIN {X 0,Y 256.136,Z 598.578,A -85,B 0,C 180,E1 -18577.279,E2 -18577.279} C_VEL
LIN {X 0,Y 256.082,Z 598.553,A -85,B 0,C 180,E1 -18581.198,E2 -18581.198} C_VEL
LIN {X 0,Y 256.094,Z 598.551,A -85,B 0,C 180,E1 -18582.329,E2 -18582.329} C_VEL
LIN {X 0,Y 257.042,Z 601.271,A -85,B 0,C 180,E1 -18582.611,E2 -18582.611} C_VEL
LIN {X 0,Y 258.851,Z 603.656,A -85,B 0,C 180,E1 -18583.039,E2 -18583.039} C_VEL
LIN {X 0,Y 261.122,Z 607.181,A -85,B 0,C 180,E1 -18583.583,E2 -18583.583} C_VEL
LIN {X 0,Y 270.381,Z 622.375,A -85,B 0,C 180,E1 -18585.685,E2 -18585.685} C_VEL
LIN {X 0,Y 278.243,Z 637.131,A -85,B 0,C 180,E1 -18587.374,E2 -18587.374} C_VEL
LIN {X 0,Y 279.342,Z 639.342,A -85,B 0,C 180,E1 -18587.604,E2 -18587.604} C_VEL
LIN {X 0,Y 277.349,Z 691.217,A -85,B 0,C 180,E1 -18588.931,E2 -18588.931} C_VEL
LIN {X 0,Y 276.628,Z 704.621,A -85,B 0,C 180,E1 -18589.507,E2 -18589.507} C_VEL
LIN {X 0,Y 275.444,Z 717.627,A -85,B 0,C 180,E1 -18590.367,E2 -18590.367} C_VEL
LIN {X 0,Y 273.67,Z 729.921,A -85,B 0,C 180,E1 -18591.484,E2 -18591.484} C_VEL
LIN {X 0,Y 271.724,Z 740.949,A -85,B 0,C 180,E1 -18592.802,E2 -18592.802} C_VEL
LIN {X 0,Y 269.6,Z 750.914,A -85,B 0,C 180,E1 -18594.299,E2 -18594.299} C_VEL
LIN {X 0,Y 267.259,Z 760.182,A -85,B 0,C 180,E1 -18596.028,E2 -18596.028} C_VEL
LIN {X 0,Y 264.9,Z 768.969,A -85,B 0,C 180,E1 -18598.102,E2 -18598.102} C_VEL
LIN {X 0,Y 262.574,Z 776.523,A -85,B 0,C 180,E1 -18600.32,E2 -18600.32} C_VEL
LIN {X 0,Y 260.479,Z 782.893,A -85,B 0,C 180,E1 -18602.699,E2 -18602.699} C_VEL
LIN {X 0,Y 258.745,Z 787.853,A -85,B 0,C 180,E1 -18605.102,E2 -18605.102} C_VEL
LIN {X 0,Y 257.383,Z 791.611,A -85,B 0,C 180,E1 -18607.526,E2 -18607.526} C_VEL
LIN {X 0,Y 256.639,Z 793.515,A -85,B 0,C 180,E1 -18609.146,E2 -18609.146} C_VEL
LIN {X 0,Y 255.964,Z 794.99,A -85,B 0,C 180,E1 -18610.763,E2 -18610.763} C_VEL
LIN {X 0,Y 255.466,Z 795.986,A -85,B 0,C 180,E1 -18612.386,E2 -18612.386} C_VEL
LIN {X 0,Y 255.036,Z 796.714,A -85,B 0,C 180,E1 -18614.687,E2 -18614.687} C_VEL
LIN {X 0,Y 254.693,Z 796.546,A -85,B 0,C 180,E1 -18617.247,E2 -18617.247} C_VEL
LIN {X 0,Y 254.697,Z 794.874,A -85,B 0,C 180,E1 -18620.47,E2 -18620.47} C_VEL
LIN {X 0,Y 254.992,Z 792.551,A -85,B 0,C 180,E1 -18622.85,E2 -18622.85} C_VEL
LIN {X 0,Y 255.419,Z 789.197,A -85,B 0,C 180,E1 -18625.265,E2 -18625.265} C_VEL
LIN {X 0,Y 256.067,Z 784.804,A -85,B 0,C 180,E1 -18627.641,E2 -18627.641} C_VEL
LIN {X 0,Y 257.111,Z 778.131,A -85,B 0,C 180,E1 -18630.392,E2 -18630.392} C_VEL
LIN {X 0,Y 258.301,Z 770.881,A -85,B 0,C 180,E1 -18632.729,E2 -18632.729} C_VEL
LIN {X 0,Y 259.605,Z 763.467,A -85,B 0,C 180,E1 -18634.658,E2 -18634.658} C_VEL
LIN {X 0,Y 261.074,Z 754.499,A -85,B 0,C 180,E1 -18636.569,E2 -18636.569} C_VEL
LIN {X 0,Y 262.47,Z 744.578,A -85,B 0,C 180,E1 -18638.275,E2 -18638.275} C_VEL
LIN {X 0,Y 264.055,Z 732.705,A -85,B 0,C 180,E1 -18639.885,E2 -18639.885} C_VEL
LIN {X 0,Y 265.279,Z 721.37,A -85,B 0,C 180,E1 -18641.067,E2 -18641.067} C_VEL
LIN {X 0,Y 266.268,Z 708.199,A -85,B 0,C 180,E1 -18642.087,E2 -18642.087} C_VEL
LIN {X 0,Y 266.884,Z 695.749,A -85,B 0,C 180,E1 -18642.748,E2 -18642.748} C_VEL
LIN {X 0,Y 267.621,Z 668.491,A -85,B 0,C 180,E1 -18643.528,E2 -18643.528} C_VEL
LIN {X 0,Y 268.699,Z 628.014,A -85,B 0,C 180,E1 -18644.588,E2 -18644.588} C_VEL
LIN {X 0,Y 259.733,Z 606.591,A -85,B 0,C 180,E1 -18646.055,E2 -18646.055} C_VEL
LIN {X 0,Y 256.44,Z 599.436,A -85,B 0,C 180,E1 -18646.602,E2 -18646.602} C_VEL
LIN {X 0,Y 256.276,Z 598.563,A -85,B 0,C 180,E1 -18646.66,E2 -18646.66} C_VEL
LIN {X 0,Y 256.24,Z 598.567,A -85,B 0,C 180,E1 -18646.963,E2 -18646.963} C_VEL
LIN {X 0,Y 257.718,Z 602.591,A -85,B 0,C 180,E1 -18647.257,E2 -18647.257} C_VEL
LIN {X 0,Y 267.78,Z 626.226,A -85,B 0,C 180,E1 -18648.971,E2 -18648.971} C_VEL
LIN {X 0,Y 269.337,Z 630.125,A -85,B 0,C 180,E1 -18649.234,E2 -18649.234} C_VEL
LIN {X 0,Y 267.163,Z 692.832,A -85,B 0,C 180,E1 -18651.121,E2 -18651.121} C_VEL
LIN {X 0,Y 266.57,Z 706.145,A -85,B 0,C 180,E1 -18651.816,E2 -18651.816} C_VEL
LIN {X 0,Y 265.61,Z 717.964,A -85,B 0,C 180,E1 -18652.69,E2 -18652.69} C_VEL
LIN {X 0,Y 264.356,Z 730.329,A -85,B 0,C 180,E1 -18653.917,E2 -18653.917} C_VEL
LIN {X 0,Y 262.835,Z 742.759,A -85,B 0,C 180,E1 -18655.541,E2 -18655.541} C_VEL
LIN {X 0,Y 261.382,Z 752.861,A -85,B 0,C 180,E1 -18657.199,E2 -18657.199} C_VEL
LIN {X 0,Y 259.884,Z 762.311,A -85,B 0,C 180,E1 -18659.128,E2 -18659.128} C_VEL
LIN {X 0,Y 258.425,Z 771.264,A -85,B 0,C 180,E1 -18661.398,E2 -18661.398} C_VEL
LIN {X 0,Y 257.265,Z 778.013,A -85,B 0,C 180,E1 -18663.514,E2 -18663.514} C_VEL
LIN {X 0,Y 256.266,Z 784.628,A -85,B 0,C 180,E1 -18666.13,E2 -18666.13} C_VEL
LIN {X 0,Y 255.638,Z 788.785,A -85,B 0,C 180,E1 -18668.21,E2 -18668.21} C_VEL
LIN {X 0,Y 255.098,Z 792.25,A -85,B 0,C 180,E1 -18670.437,E2 -18670.437} C_VEL
LIN {X 0,Y 254.806,Z 793.998,A -85,B 0,C 180,E1 -18671.866,E2 -18671.866} C_VEL
LIN {X 0,Y 254.598,Z 796.034,A -85,B 0,C 180,E1 -18674.134,E2 -18674.134} C_VEL
LIN {X 0,Y 254.605,Z 797.194,A -85,B 0,C 180,E1 -18676.363,E2 -18676.363} C_VEL
LIN {X 0,Y 254.803,Z 797.569,A -85,B 0,C 180,E1 -18678.549,E2 -18678.549} C_VEL
LIN {X 0,Y 255.248,Z 797.201,A -85,B 0,C 180,E1 -18680.707,E2 -18680.707} C_VEL
LIN {X 0,Y 255.89,Z 796.079,A -85,B 0,C 180,E1 -18682.826,E2 -18682.826} C_VEL
LIN {X 0,Y 256.792,Z 793.939,A -85,B 0,C 180,E1 -18685.188,E2 -18685.188} C_VEL
LIN {X 0,Y 257.971,Z 790.693,A -85,B 0,C 180,E1 -18687.621,E2 -18687.621} C_VEL
LIN {X 0,Y 259.508,Z 786.23,A -85,B 0,C 180,E1 -18690.066,E2 -18690.066} C_VEL
LIN {X 0,Y 261.44,Z 780.358,A -85,B 0,C 180,E1 -18692.509,E2 -18692.509} C_VEL
LIN {X 0,Y 263.762,Z 772.793,A -85,B 0,C 180,E1 -18694.947,E2 -18694.947} C_VEL
LIN {X 0,Y 264.932,Z 768.79,A -85,B 0,C 180,E1 -18696.025,E2 -18696.025} C_VEL
LIN {X 0,Y 265.454,Z 765.089,A -85,B 0,C 180,E1 -18697.016,E2 -18697.016} C_VEL
LIN {X 0,Y 264.649,Z 758.962,A -85,B 0,C 180,E1 -18698.697,E2 -18698.697} C_VEL
LIN {X 0,Y 263.826,Z 752.296,A -85,B 0,C 180,E1 -18700.276,E2 -18700.276} C_VEL
LIN {X 0,Y 264.28,Z 747.756,A -85,B 0,C 180,E1 -18701.087,E2 -18701.087} C_VEL
LIN {X 0,Y 266.493,Z 737.049,A -85,B 0,C 180,E1 -18702.56,E2 -18702.56} C_VEL
LIN {X 0,Y 268.395,Z 725.642,A -85,B 0,C 180,E1 -18703.797,E2 -18703.797} C_VEL
LIN {X 0,Y 269.981,Z 713.034,A -85,B 0,C 180,E1 -18704.833,E2 -18704.833} C_VEL
LIN {X 0,Y 271.004,Z 700.635,A -85,B 0,C 180,E1 -18705.557,E2 -18705.557} C_VEL
LIN {X 0,Y 271.865,Z 683.962,A -85,B 0,C 180,E1 -18706.16,E2 -18706.16} C_VEL
LIN {X 0,Y 274.299,Z 641.182,A -85,B 0,C 180,E1 -18707.467,E2 -18707.467} C_VEL
LIN {X 0,Y 267.74,Z 628.283,A -85,B 0,C 180,E1 -18709.267,E2 -18709.267} C_VEL
LIN {X 0,Y 260.509,Z 616.403,A -85,B 0,C 180,E1 -18711.369,E2 -18711.369} C_VEL
LIN {X 0,Y 257.332,Z 611.602,A -85,B 0,C 180,E1 -18712.349,E2 -18712.349} C_VEL
LIN {X 0,Y 255.351,Z 608.627,A -85,B 0,C 180,E1 -18712.995,E2 -18712.995} C_VEL
LIN {X 0,Y 253.194,Z 605.513,A -85,B 0,C 180,E1 -18713.725,E2 -18713.725} C_VEL
LIN {X 0,Y 252.688,Z 604.543,A -85,B 0,C 180,E1 -18713.913,E2 -18713.913} C_VEL
LIN {X 0,Y 250.514,Z 602.541,A -85,B 0,C 180,E1 -18714.617,E2 -18714.617} C_VEL
LIN {X 0,Y 249.448,Z 600.138,A -85,B 0,C 180,E1 -18715.05,E2 -18715.05} C_VEL
LIN {X 0,Y 249.311,Z 599.426,A -85,B 0,C 180,E1 -18715.149,E2 -18715.149} C_VEL
LIN {X 0,Y 249.671,Z 599.382,A -85,B 0,C 180,E1 -18718.387,E2 -18718.387} C_VEL
LIN {X 0,Y 249.671,Z 599.384,A -85,B 0,C 180,E1 -18721.613,E2 -18721.613} C_VEL
LIN {X 0,Y 249.455,Z 599.402,A -85,B 0,C 180,E1 -18726.471,E2 -18726.471} C_VEL
LIN {X 0,Y 249.384,Z 599.408,A -85,B 0,C 180,E1 -18729.735,E2 -18729.735} C_VEL
LIN {X 0,Y 249.192,Z 599.433,A -85,B 0,C 180,E1 -18734.704,E2 -18734.704} C_VEL
LIN {X 0,Y 249.13,Z 599.442,A -85,B 0,C 180,E1 -18738.078,E2 -18738.078} C_VEL
LIN {X 0,Y 249.082,Z 599.45,A -85,B 0,C 180,E1 -18741.519,E2 -18741.519} C_VEL
LIN {X 0,Y 249.126,Z 599.453,A -85,B 0,C 180,E1 -18745.483,E2 -18745.483} C_VEL
LIN {X 0,Y 249.079,Z 599.46,A -85,B 0,C 180,E1 -18748.994,E2 -18748.994} C_VEL
LIN {X 0,Y 249.032,Z 599.465,A -85,B 0,C 180,E1 -18752.426,E2 -18752.426} C_VEL
LIN {X 0,Y 249.072,Z 599.454,A -85,B 0,C 180,E1 -18756.338,E2 -18756.338} C_VEL
LIN {X 0,Y 249.077,Z 599.507,A -85,B 0,C 180,E1 -18760.998,E2 -18760.998} C_VEL
LIN {X 0,Y 251.539,Z 607.272,A -85,B 0,C 180,E1 -18765.695,E2 -18765.695} C_VEL
LIN {X 0,Y 253.484,Z 613.695,A -85,B 0,C 180,E1 -18769.032,E2 -18769.032} C_VEL
LIN {X 0,Y 255.278,Z 620.736,A -85,B 0,C 180,E1 -18772.251,E2 -18772.251} C_VEL
LIN {X 0,Y 258.025,Z 625.972,A -85,B 0,C 180,E1 -18773.172,E2 -18773.172} C_VEL
LIN {X 0,Y 261.995,Z 634.008,A -85,B 0,C 180,E1 -18774.451,E2 -18774.451} C_VEL
LIN {X 0,Y 266.268,Z 643.226,A -85,B 0,C 180,E1 -18775.747,E2 -18775.747} C_VEL
LIN {X 0,Y 267.455,Z 646.426,A -85,B 0,C 180,E1 -18776.12,E2 -18776.12} C_VEL
LIN {X 0,Y 270.142,Z 665.674,A -85,B 0,C 180,E1 -18777.449,E2 -18777.449} C_VEL
LIN {X 0,Y 271.585,Z 681.293,A -85,B 0,C 180,E1 -18778.336,E2 -18778.336} C_VEL
LIN {X 0,Y 272.124,Z 690.345,A -85,B 0,C 180,E1 -18778.79,E2 -18778.79} C_VEL
LIN {X 0,Y 269.613,Z 734.269,A -85,B 0,C 180,E1 -18780.164,E2 -18780.164} C_VEL
LIN {X 0,Y 268.084,Z 748.305,A -85,B 0,C 180,E1 -18780.882,E2 -18780.882} C_VEL
LIN {X 0,Y 266.019,Z 761.087,A -85,B 0,C 180,E1 -18781.821,E2 -18781.821} C_VEL
LIN {X 0,Y 263.511,Z 773.361,A -85,B 0,C 180,E1 -18783.039,E2 -18783.039} C_VEL
LIN {X 0,Y 260.875,Z 784.54,A -85,B 0,C 180,E1 -18784.467,E2 -18784.467} C_VEL
LIN {X 0,Y 257.977,Z 795.708,A -85,B 0,C 180,E1 -18786.308,E2 -18786.308} C_VEL
LIN {X 0,Y 255.394,Z 804.839,A -85,B 0,C 180,E1 -18788.193,E2 -18788.193} C_VEL
LIN {X 0,Y 252.889,Z 813.843,A -85,B 0,C 180,E1 -18790.52,E2 -18790.52} C_VEL
LIN {X 0,Y 250.977,Z 821.114,A -85,B 0,C 180,E1 -18792.901,E2 -18792.901} C_VEL
LIN {X 0,Y 249.306,Z 827.013,A -85,B 0,C 180,E1 -18795.303,E2 -18795.303} C_VEL
LIN {X 0,Y 248.096,Z 831.736,A -85,B 0,C 180,E1 -18797.734,E2 -18797.734} C_VEL
LIN {X 0,Y 247.523,Z 835.398,A -85,B 0,C 180,E1 -18800.192,E2 -18800.192} C_VEL
LIN {X 0,Y 247.272,Z 838.73,A -85,B 0,C 180,E1 -18803.472,E2 -18803.472} C_VEL
LIN {X 0,Y 247.332,Z 839.784,A -85,B 0,C 180,E1 -18805.11,E2 -18805.11} C_VEL
LIN {X 0,Y 247.691,Z 840.591,A -85,B 0,C 180,E1 -18808.374,E2 -18808.374} C_VEL
LIN {X 0,Y 247.815,Z 840.373,A -85,B 0,C 180,E1 -18810,E2 -18810} C_VEL
LIN {X 0,Y 247.761,Z 839.715,A -85,B 0,C 180,E1 -18811.625,E2 -18811.625} C_VEL
LIN {X 0,Y 247.309,Z 838.202,A -85,B 0,C 180,E1 -18815.941,E2 -18815.941} C_VEL
LIN {X 0,Y 247.283,Z 836.523,A -85,B 0,C 180,E1 -18818.169,E2 -18818.169} C_VEL
LIN {X 0,Y 247.68,Z 833.783,A -85,B 0,C 180,E1 -18820.628,E2 -18820.628} C_VEL
LIN {X 0,Y 248.444,Z 830.038,A -85,B 0,C 180,E1 -18823.079,E2 -18823.079} C_VEL
LIN {X 0,Y 249.766,Z 825.197,A -85,B 0,C 180,E1 -18825.504,E2 -18825.504} C_VEL
LIN {X 0,Y 251.533,Z 819.111,A -85,B 0,C 180,E1 -18827.899,E2 -18827.899} C_VEL
LIN {X 0,Y 253.606,Z 811.578,A -85,B 0,C 180,E1 -18830.267,E2 -18830.267} C_VEL
LIN {X 0,Y 255.917,Z 803.928,A -85,B 0,C 180,E1 -18832.185,E2 -18832.185} C_VEL
LIN {X 0,Y 258.555,Z 794.633,A -85,B 0,C 180,E1 -18834.061,E2 -18834.061} C_VEL
LIN {X 0,Y 261.202,Z 784.328,A -85,B 0,C 180,E1 -18835.712,E2 -18835.712} C_VEL
LIN {X 0,Y 263.815,Z 772.919,A -85,B 0,C 180,E1 -18837.142,E2 -18837.142} C_VEL
LIN {X 0,Y 266.155,Z 760.901,A -85,B 0,C 180,E1 -18838.271,E2 -18838.271} C_VEL
LIN {X 0,Y 268.143,Z 747.624,A -85,B 0,C 180,E1 -18839.165,E2 -18839.165} C_VEL
LIN {X 0,Y 269.358,Z 734.608,A -85,B 0,C 180,E1 -18839.752,E2 -18839.752} C_VEL
LIN {X 0,Y 271.292,Z 685.607,A -85,B 0,C 180,E1 -18841.074,E2 -18841.074} C_VEL
LIN {X 0,Y 269.087,Z 660.599,A -85,B 0,C 180,E1 -18842.222,E2 -18842.222} C_VEL
LIN {X 0,Y 266.563,Z 641.019,A -85,B 0,C 180,E1 -18843.275,E2 -18843.275} C_VEL
LIN {X 0,Y 258.806,Z 621.965,A -85,B 0,C 180,E1 -18845.277,E2 -18845.277} C_VEL
LIN {X 0,Y 255.188,Z 613.724,A -85,B 0,C 180,E1 -18846.265,E2 -18846.265} C_VEL
LIN {X 0,Y 252.263,Z 605.947,A -85,B 0,C 180,E1 -18847.522,E2 -18847.522} C_VEL
LIN {X 0,Y 250.841,Z 603.293,A -85,B 0,C 180,E1 -18848.052,E2 -18848.052} C_VEL
LIN {X 0,Y 249.299,Z 600.577,A -85,B 0,C 180,E1 -18848.634,E2 -18848.634} C_VEL
LIN {X 0,Y 249.065,Z 599.452,A -85,B 0,C 180,E1 -18848.824,E2 -18848.824} C_VEL
LIN {X 0,Y 249.044,Z 599.456,A -85,B 0,C 180,E1 -18852.801,E2 -18852.801} C_VEL
LIN {X 0,Y 249.06,Z 599.46,A -85,B 0,C 180,E1 -18857.372,E2 -18857.372} C_VEL
LIN {X 0,Y 249.05,Z 599.455,A -85,B 0,C 180,E1 -18861.624,E2 -18861.624} C_VEL
LIN {X 0,Y 249.058,Z 599.442,A -85,B 0,C 180,E1 -18865.642,E2 -18865.642} C_VEL
LIN {X 0,Y 249.044,Z 599.453,A -85,B 0,C 180,E1 -18869.472,E2 -18869.472} C_VEL
LIN {X 0,Y 249.068,Z 599.456,A -85,B 0,C 180,E1 -18873.162,E2 -18873.162} C_VEL
LIN {X 0,Y 249.074,Z 599.436,A -85,B 0,C 180,E1 -18876.732,E2 -18876.732} C_VEL
LIN {X 0,Y 249.106,Z 599.454,A -85,B 0,C 180,E1 -18880.211,E2 -18880.211} C_VEL
LIN {X 0,Y 249.218,Z 599.416,A -85,B 0,C 180,E1 -18883.62,E2 -18883.62} C_VEL
LIN {X 0,Y 249.238,Z 599.433,A -85,B 0,C 180,E1 -18888.616,E2 -18888.616} C_VEL
LIN {X 0,Y 249.449,Z 599.387,A -85,B 0,C 180,E1 -18891.902,E2 -18891.902} C_VEL
LIN {X 0,Y 249.294,Z 599.431,A -85,B 0,C 180,E1 -18895.148,E2 -18895.148} C_VEL
LIN {X 0,Y 249.671,Z 599.357,A -85,B 0,C 180,E1 -18898.387,E2 -18898.387} C_VEL
LIN {X 0,Y 249.673,Z 599.384,A -85,B 0,C 180,E1 -18901.613,E2 -18901.613} C_VEL
LIN {X 0,Y 249.443,Z 599.39,A -85,B 0,C 180,E1 -18906.727,E2 -18906.727} C_VEL
LIN {X 0,Y 249.384,Z 599.419,A -85,B 0,C 180,E1 -18909.735,E2 -18909.735} C_VEL
LIN {X 0,Y 249.199,Z 599.438,A -85,B 0,C 180,E1 -18914.704,E2 -18914.704} C_VEL
LIN {X 0,Y 249.134,Z 599.434,A -85,B 0,C 180,E1 -18918.078,E2 -18918.078} C_VEL
